LIN {X 0,Y 299.313,Z 470.406,A -85,B 0,C 180,E1 -16726.074,E2 -16726.074} C_VEL
LIN {X 0,Y 297.417,Z 475.338,A -85,B 0,C 180,E1 -16727.721,E2 -16727.721} C_VEL
LIN {X 0,Y 295.4,Z 479.817,A -85,B 0,C 180,E1 -16729.721,E2 -16729.721} C_VEL
LIN {X 0,Y 293.632,Z 482.84,A -85,B 0,C 180,E1 -16731.743,E2 -16731.743} C_VEL
LIN {X 0,Y 292.623,Z 484.058,A -85,B 0,C 180,E1 -16733.103,E2 -16733.103} C_VEL
LIN {X 0,Y 291.792,Z 484.661,A -85,B 0,C 180,E1 -16734.471,E2 -16734.471} C_VEL
LIN {X 0,Y 291.126,Z 484.675,A -85,B 0,C 180,E1 -16735.847,E2 -16735.847} C_VEL
LIN {X 0,Y 290.687,Z 484.067,A -85,B 0,C 180,E1 -16737.229,E2 -16737.229} C_VEL
LIN {X 0,Y 290.38,Z 482.836,A -85,B 0,C 180,E1 -16738.613,E2 -16738.613} C_VEL
LIN {X 0,Y 290.157,Z 479.788,A -85,B 0,C 180,E1 -16740.694,E2 -16740.694} C_VEL
LIN {X 0,Y 290.14,Z 475.202,A -85,B 0,C 180,E1 -16742.777,E2 -16742.777} C_VEL
LIN {X 0,Y 290.478,Z 468.838,A -85,B 0,C 180,E1 -16744.858,E2 -16744.858} C_VEL
LIN {X 0,Y 290.817,Z 461.925,A -85,B 0,C 180,E1 -16746.592,E2 -16746.592} C_VEL
LIN {X 0,Y 291.139,Z 453.117,A -85,B 0,C 180,E1 -16748.328,E2 -16748.328} C_VEL
LIN {X 0,Y 291.598,Z 443.01,A -85,B 0,C 180,E1 -16749.888,E2 -16749.888} C_VEL
LIN {X 0,Y 292.119,Z 433.031,A -85,B 0,C 180,E1 -16751.097,E2 -16751.097} C_VEL
LIN {X 0,Y 290.871,Z 421.3,A -85,B 0,C 180,E1 -16752.206,E2 -16752.206} C_VEL
LIN {X 0,Y 290.218,Z 413.705,A -85,B 0,C 180,E1 -16752.766,E2 -16752.766} C_VEL
LIN {X 0,Y 290.434,Z 407.138,A -85,B 0,C 180,E1 -16756.881,E2 -16756.881} C_VEL
LIN {X 0,Y 290.756,Z 401.449,A -85,B 0,C 180,E1 -16760.517,E2 -16760.517} C_VEL
LIN {X 0,Y 291.158,Z 394.62,A -85,B 0,C 180,E1 -16764.987,E2 -16764.987} C_VEL
LIN {X 0,Y 291.612,Z 388.864,A -85,B 0,C 180,E1 -16768.817,E2 -16768.817} C_VEL
LIN {X 0,Y 291.797,Z 385.393,A -85,B 0,C 180,E1 -16771.187,E2 -16771.187} C_VEL
LIN {X 0,Y 291.576,Z 384.166,A -85,B 0,C 180,E1 -16772.181,E2 -16772.181} C_VEL
LIN {X 0,Y 291.408,Z 384.187,A -85,B 0,C 180,E1 -16777.081,E2 -16777.081} C_VEL
LIN {X 0,Y 291.335,Z 384.196,A -85,B 0,C 180,E1 -16780.642,E2 -16780.642} C_VEL
LIN {X 0,Y 291.316,Z 384.196,A -85,B 0,C 180,E1 -16784.397,E2 -16784.397} C_VEL
LIN {X 0,Y 291.33,Z 384.196,A -85,B 0,C 180,E1 -16788.404,E2 -16788.404} C_VEL
LIN {X 0,Y 291.35,Z 384.191,A -85,B 0,C 180,E1 -16791.158,E2 -16791.158} C_VEL
LIN {X 0,Y 291.364,Z 384.194,A -85,B 0,C 180,E1 -16794.626,E2 -16794.626} C_VEL
LIN {X 0,Y 291.373,Z 384.188,A -85,B 0,C 180,E1 -16797.951,E2 -16797.951} C_VEL
LIN {X 0,Y 291.38,Z 384.187,A -85,B 0,C 180,E1 -16801.158,E2 -16801.158} C_VEL
LIN {X 0,Y 291.418,Z 384.186,A -85,B 0,C 180,E1 -16804.272,E2 -16804.272} C_VEL
LIN {X 0,Y 291.392,Z 384.185,A -85,B 0,C 180,E1 -16807.3,E2 -16807.3} C_VEL
LIN {X 0,Y 291.462,Z 384.18,A -85,B 0,C 180,E1 -16810.27,E2 -16810.27} C_VEL
LIN {X 0,Y 291.558,Z 384.166,A -85,B 0,C 180,E1 -16814.624,E2 -16814.624} C_VEL
LIN {X 0,Y 291.539,Z 384.167,A -85,B 0,C 180,E1 -16818.881,E2 -16818.881} C_VEL
LIN {X 0,Y 291.691,Z 384.15,A -85,B 0,C 180,E1 -16821.688,E2 -16821.688} C_VEL
LIN {X 0,Y 291.63,Z 384.157,A -85,B 0,C 180,E1 -16824.468,E2 -16824.468} C_VEL
LIN {X 0,Y 291.892,Z 384.124,A -85,B 0,C 180,E1 -16828.62,E2 -16828.62} C_VEL
LIN {X 0,Y 291.894,Z 384.124,A -85,B 0,C 180,E1 -16831.38,E2 -16831.38} C_VEL
LIN {X 0,Y 291.745,Z 384.141,A -85,B 0,C 180,E1 -16836.918,E2 -16836.918} C_VEL
LIN {X 0,Y 291.632,Z 384.159,A -85,B 0,C 180,E1 -16839.712,E2 -16839.712} C_VEL
LIN {X 0,Y 291.525,Z 384.172,A -85,B 0,C 180,E1 -16843.95,E2 -16843.95} C_VEL
LIN {X 0,Y 291.49,Z 384.173,A -85,B 0,C 180,E1 -16846.818,E2 -16846.818} C_VEL
LIN {X 0,Y 291.454,Z 384.18,A -85,B 0,C 180,E1 -16849.875,E2 -16849.875} C_VEL
LIN {X 0,Y 291.403,Z 384.185,A -85,B 0,C 180,E1 -16854.205,E2 -16854.205} C_VEL
LIN {X 0,Y 291.422,Z 384.184,A -85,B 0,C 180,E1 -16857.272,E2 -16857.272} C_VEL
LIN {X 0,Y 291.336,Z 384.191,A -85,B 0,C 180,E1 -16860.437,E2 -16860.437} C_VEL
LIN {X 0,Y 291.347,Z 384.194,A -85,B 0,C 180,E1 -16863.698,E2 -16863.698} C_VEL
LIN {X 0,Y 291.397,Z 384.188,A -85,B 0,C 180,E1 -16867.259,E2 -16867.259} C_VEL
LIN {X 0,Y 291.336,Z 384.192,A -85,B 0,C 180,E1 -16870.642,E2 -16870.642} C_VEL
LIN {X 0,Y 291.291,Z 384.198,A -85,B 0,C 180,E1 -16874.402,E2 -16874.402} C_VEL
LIN {X 0,Y 291.328,Z 384.193,A -85,B 0,C 180,E1 -16878.404,E2 -16878.404} C_VEL
LIN {X 0,Y 291.35,Z 384.196,A -85,B 0,C 180,E1 -16881.157,E2 -16881.157} C_VEL
LIN {X 0,Y 291.362,Z 384.19,A -85,B 0,C 180,E1 -16884.626,E2 -16884.626} C_VEL
LIN {X 0,Y 291.374,Z 384.187,A -85,B 0,C 180,E1 -16887.951,E2 -16887.951} C_VEL
LIN {X 0,Y 291.385,Z 384.189,A -85,B 0,C 180,E1 -16891.158,E2 -16891.158} C_VEL
LIN {X 0,Y 291.418,Z 384.182,A -85,B 0,C 180,E1 -16894.272,E2 -16894.272} C_VEL
LIN {X 0,Y 291.384,Z 384.188,A -85,B 0,C 180,E1 -16897.3,E2 -16897.3} C_VEL
LIN {X 0,Y 291.46,Z 384.178,A -85,B 0,C 180,E1 -16900.27,E2 -16900.27} C_VEL
LIN {X 0,Y 291.557,Z 384.168,A -85,B 0,C 180,E1 -16904.624,E2 -16904.624} C_VEL
LIN {X 0,Y 291.541,Z 384.17,A -85,B 0,C 180,E1 -16908.881,E2 -16908.881} C_VEL
LIN {X 0,Y 291.711,Z 384.144,A -85,B 0,C 180,E1 -16911.688,E2 -16911.688} C_VEL
LIN {X 0,Y 291.633,Z 384.159,A -85,B 0,C 180,E1 -16914.468,E2 -16914.468} C_VEL
LIN {X 0,Y 291.892,Z 384.126,A -85,B 0,C 180,E1 -16918.62,E2 -16918.62} C_VEL
LIN {X 0,Y 291.895,Z 384.122,A -85,B 0,C 180,E1 -16921.38,E2 -16921.38} C_VEL
LIN {X 0,Y 291.749,Z 384.141,A -85,B 0,C 180,E1 -16926.918,E2 -16926.918} C_VEL
LIN {X 0,Y 291.631,Z 384.155,A -85,B 0,C 180,E1 -16929.712,E2 -16929.712} C_VEL
LIN {X 0,Y 291.502,Z 384.172,A -85,B 0,C 180,E1 -16933.035,E2 -16933.035} C_VEL
LIN {X 0,Y 290.827,Z 384.26,A -85,B 0,C 180,E1 -16934.188,E2 -16934.188} C_VEL
LIN {X 0,Y 287.966,Z 384.615,A -85,B 0,C 180,E1 -16936.065,E2 -16936.065} C_VEL
LIN {X 0,Y 285.533,Z 384.917,A -85,B 0,C 180,E1 -16937.589,E2 -16937.589} C_VEL
LIN {X 0,Y 284.476,Z 385.048,A -85,B 0,C 180,E1 -16938.77,E2 -16938.77} C_VEL
LIN {X 0,Y 284.383,Z 385.058,A -85,B 0,C 180,E1 -16939.171,E2 -16939.171} C_VEL
LIN {X 0,Y 284.371,Z 385.063,A -85,B 0,C 180,E1 -16943.875,E2 -16943.875} C_VEL
LIN {X 0,Y 284.397,Z 385.056,A -85,B 0,C 180,E1 -16947.173,E2 -16947.173} C_VEL
LIN {X 0,Y 284.295,Z 385.07,A -85,B 0,C 180,E1 -16951.274,E2 -16951.274} C_VEL
LIN {X 0,Y 284.363,Z 385.061,A -85,B 0,C 180,E1 -16955.354,E2 -16955.354} C_VEL
LIN {X 0,Y 284.325,Z 385.068,A -85,B 0,C 180,E1 -16958.167,E2 -16958.167} C_VEL
LIN {X 0,Y 284.271,Z 385.073,A -85,B 0,C 180,E1 -16962.125,E2 -16962.125} C_VEL
LIN {X 0,Y 284.287,Z 385.073,A -85,B 0,C 180,E1 -16966.195,E2 -16966.195} C_VEL
LIN {X 0,Y 284.354,Z 385.245,A -85,B 0,C 180,E1 -16968.499,E2 -16968.499} C_VEL
LIN {X 0,Y 286.142,Z 394.145,A -85,B 0,C 180,E1 -16972.563,E2 -16972.563} C_VEL
LIN {X 0,Y 288.209,Z 404.002,A -85,B 0,C 180,E1 -16976.866,E2 -16976.866} C_VEL
LIN {X 0,Y 289.225,Z 409.855,A -85,B 0,C 180,E1 -16979.317,E2 -16979.317} C_VEL
LIN {X 0,Y 286.887,Z 421.364,A -85,B 0,C 180,E1 -16983.835,E2 -16983.835} C_VEL
LIN {X 0,Y 284.814,Z 434.601,A -85,B 0,C 180,E1 -16989.035,E2 -16989.035} C_VEL
LIN {X 0,Y 284.356,Z 438.709,A -85,B 0,C 180,E1 -16990.65,E2 -16990.65} C_VEL
LIN {X 0,Y 284.635,Z 450.827,A -85,B 0,C 180,E1 -16991.277,E2 -16991.277} C_VEL
LIN {X 0,Y 285.426,Z 463.008,A -85,B 0,C 180,E1 -16992.167,E2 -16992.167} C_VEL
LIN {X 0,Y 286.069,Z 473.069,A -85,B 0,C 180,E1 -16993.126,E2 -16993.126} C_VEL
LIN {X 0,Y 285.367,Z 484.226,A -85,B 0,C 180,E1 -16994.465,E2 -16994.465} C_VEL
LIN {X 0,Y 284.62,Z 493.685,A -85,B 0,C 180,E1 -16995.887,E2 -16995.887} C_VEL
LIN {X 0,Y 284.078,Z 502.385,A -85,B 0,C 180,E1 -16997.498,E2 -16997.498} C_VEL
LIN {X 0,Y 283.619,Z 510.299,A -85,B 0,C 180,E1 -16999.289,E2 -16999.289} C_VEL
LIN {X 0,Y 283.365,Z 517.923,A -85,B 0,C 180,E1 -17001.442,E2 -17001.442} C_VEL
LIN {X 0,Y 283.392,Z 524.403,A -85,B 0,C 180,E1 -17003.804,E2 -17003.804} C_VEL
LIN {X 0,Y 283.412,Z 528.421,A -85,B 0,C 180,E1 -17005.734,E2 -17005.734} C_VEL
LIN {X 0,Y 283.463,Z 530.725,A -85,B 0,C 180,E1 -17007.158,E2 -17007.158} C_VEL
LIN {X 0,Y 283.429,Z 532.5,A -85,B 0,C 180,E1 -17008.579,E2 -17008.579} C_VEL
LIN {X 0,Y 283.353,Z 533.796,A -85,B 0,C 180,E1 -17010,E2 -17010} C_VEL
LIN {X 0,Y 283.316,Z 534.601,A -85,B 0,C 180,E1 -17011.422,E2 -17011.422} C_VEL
LIN {X 0,Y 283.067,Z 534.958,A -85,B 0,C 180,E1 -17012.846,E2 -17012.846} C_VEL
LIN {X 0,Y 282.807,Z 534.888,A -85,B 0,C 180,E1 -17014.276,E2 -17014.276} C_VEL
LIN {X 0,Y 282.714,Z 534.18,A -85,B 0,C 180,E1 -17016.087,E2 -17016.087} C_VEL
LIN {X 0,Y 282.793,Z 532.167,A -85,B 0,C 180,E1 -17018.576,E2 -17018.576} C_VEL
LIN {X 0,Y 283.348,Z 528.257,A -85,B 0,C 180,E1 -17021.445,E2 -17021.445} C_VEL
LIN {X 0,Y 284.44,Z 524.2,A -85,B 0,C 180,E1 -17023.576,E2 -17023.576} C_VEL
LIN {X 0,Y 285.821,Z 519.069,A -85,B 0,C 180,E1 -17025.693,E2 -17025.693} C_VEL
LIN {X 0,Y 288.032,Z 511.787,A -85,B 0,C 180,E1 -17028.043,E2 -17028.043} C_VEL
LIN {X 0,Y 290.656,Z 503.511,A -85,B 0,C 180,E1 -17030.155,E2 -17030.155} C_VEL
LIN {X 0,Y 293.667,Z 493.625,A -85,B 0,C 180,E1 -17032.144,E2 -17032.144} C_VEL
LIN {X 0,Y 296.144,Z 484.696,A -85,B 0,C 180,E1 -17033.608,E2 -17033.608} C_VEL
LIN {X 0,Y 297.823,Z 474.304,A -85,B 0,C 180,E1 -17035.136,E2 -17035.136} C_VEL
LIN {X 0,Y 298.035,Z 463.954,A -85,B 0,C 180,E1 -17036.618,E2 -17036.618} C_VEL
LIN {X 0,Y 297.261,Z 453.783,A -85,B 0,C 180,E1 -17038.065,E2 -17038.065} C_VEL
LIN {X 0,Y 295.282,Z 442.412,A -85,B 0,C 180,E1 -17039.714,E2 -17039.714} C_VEL
LIN {X 0,Y 293.524,Z 434.527,A -85,B 0,C 180,E1 -17040.894,E2 -17040.894} C_VEL
LIN {X 0,Y 294.835,Z 431.545,A -85,B 0,C 180,E1 -17042.435,E2 -17042.435} C_VEL
LIN {X 0,Y 295.09,Z 429.766,A -85,B 0,C 180,E1 -17043.532,E2 -17043.532} C_VEL
LIN {X 0,Y 294.427,Z 425.778,A -85,B 0,C 180,E1 -17046.638,E2 -17046.638} C_VEL
LIN {X 0,Y 293.633,Z 422.199,A -85,B 0,C 180,E1 -17050.259,E2 -17050.259} C_VEL
LIN {X 0,Y 293.026,Z 419.56,A -85,B 0,C 180,E1 -17054.071,E2 -17054.071} C_VEL
LIN {X 0,Y 292.456,Z 418.155,A -85,B 0,C 180,E1 -17057.711,E2 -17057.711} C_VEL
LIN {X 0,Y 292.088,Z 417.72,A -85,B 0,C 180,E1 -17061.274,E2 -17061.274} C_VEL
LIN {X 0,Y 291.76,Z 418.132,A -85,B 0,C 180,E1 -17064.682,E2 -17064.682} C_VEL
LIN {X 0,Y 291.278,Z 419.282,A -85,B 0,C 180,E1 -17067.939,E2 -17067.939} C_VEL
LIN {X 0,Y 290.309,Z 421.098,A -85,B 0,C 180,E1 -17071.042,E2 -17071.042} C_VEL
LIN {X 0,Y 289.414,Z 422.981,A -85,B 0,C 180,E1 -17073.484,E2 -17073.484} C_VEL
LIN {X 0,Y 290.356,Z 425.753,A -85,B 0,C 180,E1 -17074.171,E2 -17074.171} C_VEL
LIN {X 0,Y 292.047,Z 429.532,A -85,B 0,C 180,E1 -17075.232,E2 -17075.232} C_VEL
LIN {X 0,Y 294.97,Z 437.823,A -85,B 0,C 180,E1 -17077.353,E2 -17077.353} C_VEL
LIN {X 0,Y 297.063,Z 446.831,A -85,B 0,C 180,E1 -17079.51,E2 -17079.51} C_VEL
LIN {X 0,Y 297.877,Z 454.634,A -85,B 0,C 180,E1 -17081.366,E2 -17081.366} C_VEL
LIN {X 0,Y 297.878,Z 457.869,A -85,B 0,C 180,E1 -17082.139,E2 -17082.139} C_VEL
LIN {X 0,Y 295.496,Z 465.423,A -85,B 0,C 180,E1 -17083.772,E2 -17083.772} C_VEL
LIN {X 0,Y 292.703,Z 472.611,A -85,B 0,C 180,E1 -17085.753,E2 -17085.753} C_VEL
LIN {X 0,Y 290.705,Z 477.27,A -85,B 0,C 180,E1 -17087.433,E2 -17087.433} C_VEL
LIN {X 0,Y 288.587,Z 481.379,A -85,B 0,C 180,E1 -17089.476,E2 -17089.476} C_VEL
LIN {X 0,Y 286.711,Z 484.087,A -85,B 0,C 180,E1 -17091.543,E2 -17091.543} C_VEL
LIN {X 0,Y 285.658,Z 485.145,A -85,B 0,C 180,E1 -17092.934,E2 -17092.934} C_VEL
LIN {X 0,Y 284.788,Z 485.597,A -85,B 0,C 180,E1 -17094.335,E2 -17094.335} C_VEL
LIN {X 0,Y 284.107,Z 485.431,A -85,B 0,C 180,E1 -17095.744,E2 -17095.744} C_VEL
LIN {X 0,Y 283.625,Z 484.644,A -85,B 0,C 180,E1 -17097.159,E2 -17097.159} C_VEL
LIN {X 0,Y 283.202,Z 482.309,A -85,B 0,C 180,E1 -17099.289,E2 -17099.289} C_VEL
LIN {X 0,Y 283.014,Z 478.516,A -85,B 0,C 180,E1 -17101.423,E2 -17101.423} C_VEL
LIN {X 0,Y 283.138,Z 473.111,A -85,B 0,C 180,E1 -17103.558,E2 -17103.558} C_VEL
LIN {X 0,Y 283.491,Z 467.218,A -85,B 0,C 180,E1 -17105.334,E2 -17105.334} C_VEL
LIN {X 0,Y 283.77,Z 459.657,A -85,B 0,C 180,E1 -17107.113,E2 -17107.113} C_VEL
LIN {X 0,Y 284.156,Z 451.106,A -85,B 0,C 180,E1 -17108.713,E2 -17108.713} C_VEL
LIN {X 0,Y 284.552,Z 441.577,A -85,B 0,C 180,E1 -17110.136,E2 -17110.136} C_VEL
LIN {X 0,Y 284.985,Z 432.735,A -85,B 0,C 180,E1 -17111.198,E2 -17111.198} C_VEL
LIN {X 0,Y 283.812,Z 421.87,A -85,B 0,C 180,E1 -17112.242,E2 -17112.242} C_VEL
LIN {X 0,Y 283.147,Z 414,A -85,B 0,C 180,E1 -17112.863,E2 -17112.863} C_VEL
LIN {X 0,Y 283.379,Z 407.027,A -85,B 0,C 180,E1 -17117.314,E2 -17117.314} C_VEL
LIN {X 0,Y 283.713,Z 401.294,A -85,B 0,C 180,E1 -17121.051,E2 -17121.051} C_VEL
LIN {X 0,Y 284.077,Z 395.554,A -85,B 0,C 180,E1 -17124.871,E2 -17124.871} C_VEL
LIN {X 0,Y 284.548,Z 389.768,A -85,B 0,C 180,E1 -17128.792,E2 -17128.792} C_VEL
LIN {X 0,Y 284.772,Z 386.274,A -85,B 0,C 180,E1 -17131.216,E2 -17131.216} C_VEL
LIN {X 0,Y 284.524,Z 385.044,A -85,B 0,C 180,E1 -17132.269,E2 -17132.269} C_VEL
LIN {X 0,Y 284.343,Z 385.064,A -85,B 0,C 180,E1 -17136.385,E2 -17136.385} C_VEL
LIN {X 0,Y 284.308,Z 385.068,A -85,B 0,C 180,E1 -17139.995,E2 -17139.995} C_VEL
LIN {X 0,Y 284.268,Z 385.073,A -85,B 0,C 180,E1 -17144.195,E2 -17144.195} C_VEL
LIN {X 0,Y 284.275,Z 385.073,A -85,B 0,C 180,E1 -17148.125,E2 -17148.125} C_VEL
LIN {X 0,Y 284.322,Z 385.067,A -85,B 0,C 180,E1 -17152.279,E2 -17152.279} C_VEL
LIN {X 0,Y 284.311,Z 385.068,A -85,B 0,C 180,E1 -17155.351,E2 -17155.351} C_VEL
LIN {X 0,Y 284.296,Z 385.071,A -85,B 0,C 180,E1 -17158.726,E2 -17158.726} C_VEL
LIN {X 0,Y 284.398,Z 385.058,A -85,B 0,C 180,E1 -17162.827,E2 -17162.827} C_VEL
LIN {X 0,Y 284.372,Z 385.061,A -85,B 0,C 180,E1 -17166.707,E2 -17166.707} C_VEL
LIN {X 0,Y 284.407,Z 385.055,A -85,B 0,C 180,E1 -17171.262,E2 -17171.262} C_VEL
LIN {X 0,Y 284.495,Z 385.047,A -85,B 0,C 180,E1 -17174.459,E2 -17174.459} C_VEL
LIN {X 0,Y 284.491,Z 385.046,A -85,B 0,C 180,E1 -17178.601,E2 -17178.601} C_VEL
LIN {X 0,Y 284.642,Z 385.027,A -85,B 0,C 180,E1 -17181.48,E2 -17181.48} C_VEL
LIN {X 0,Y 284.6,Z 385.033,A -85,B 0,C 180,E1 -17184.331,E2 -17184.331} C_VEL
LIN {X 0,Y 284.858,Z 385,A -85,B 0,C 180,E1 -17188.586,E2 -17188.586} C_VEL
LIN {X 0,Y 284.859,Z 385,A -85,B 0,C 180,E1 -17191.414,E2 -17191.414} C_VEL
LIN {X 0,Y 284.697,Z 385.019,A -85,B 0,C 180,E1 -17197.09,E2 -17197.09} C_VEL
LIN {X 0,Y 284.57,Z 385.039,A -85,B 0,C 180,E1 -17199.955,E2 -17199.955} C_VEL
LIN {X 0,Y 284.485,Z 385.046,A -85,B 0,C 180,E1 -17204.303,E2 -17204.303} C_VEL
LIN {X 0,Y 284.429,Z 385.054,A -85,B 0,C 180,E1 -17207.248,E2 -17207.248} C_VEL
LIN {X 0,Y 284.384,Z 385.058,A -85,B 0,C 180,E1 -17210.242,E2 -17210.242} C_VEL
LIN {X 0,Y 284.372,Z 385.062,A -85,B 0,C 180,E1 -17213.875,E2 -17213.875} C_VEL
LIN {X 0,Y 284.397,Z 385.059,A -85,B 0,C 180,E1 -17217.173,E2 -17217.173} C_VEL
LIN {X 0,Y 284.296,Z 385.071,A -85,B 0,C 180,E1 -17221.274,E2 -17221.274} C_VEL
LIN {X 0,Y 284.364,Z 385.065,A -85,B 0,C 180,E1 -17225.354,E2 -17225.354} C_VEL
LIN {X 0,Y 284.325,Z 385.064,A -85,B 0,C 180,E1 -17228.167,E2 -17228.167} C_VEL
LIN {X 0,Y 284.271,Z 385.072,A -85,B 0,C 180,E1 -17232.124,E2 -17232.124} C_VEL
LIN {X 0,Y 284.256,Z 385.073,A -85,B 0,C 180,E1 -17236.189,E2 -17236.189} C_VEL
LIN {X 0,Y 284.308,Z 385.068,A -85,B 0,C 180,E1 -17240.024,E2 -17240.024} C_VEL
LIN {X 0,Y 284.332,Z 385.065,A -85,B 0,C 180,E1 -17243.614,E2 -17243.614} C_VEL
LIN {X 0,Y 284.309,Z 385.071,A -85,B 0,C 180,E1 -17247.189,E2 -17247.189} C_VEL
LIN {X 0,Y 284.361,Z 385.062,A -85,B 0,C 180,E1 -17250.376,E2 -17250.376} C_VEL
LIN {X 0,Y 284.38,Z 385.058,A -85,B 0,C 180,E1 -17253.587,E2 -17253.587} C_VEL
LIN {X 0,Y 284.368,Z 385.063,A -85,B 0,C 180,E1 -17256.707,E2 -17256.707} C_VEL
LIN {X 0,Y 284.406,Z 385.056,A -85,B 0,C 180,E1 -17261.262,E2 -17261.262} C_VEL
LIN {X 0,Y 284.494,Z 385.046,A -85,B 0,C 180,E1 -17264.459,E2 -17264.459} C_VEL
LIN {X 0,Y 284.492,Z 385.049,A -85,B 0,C 180,E1 -17268.601,E2 -17268.601} C_VEL
LIN {X 0,Y 284.661,Z 385.023,A -85,B 0,C 180,E1 -17271.481,E2 -17271.481} C_VEL
LIN {X 0,Y 284.603,Z 385.033,A -85,B 0,C 180,E1 -17274.331,E2 -17274.331} C_VEL
LIN {X 0,Y 284.858,Z 385.003,A -85,B 0,C 180,E1 -17278.586,E2 -17278.586} C_VEL
LIN {X 0,Y 284.861,Z 384.998,A -85,B 0,C 180,E1 -17281.414,E2 -17281.414} C_VEL
LIN {X 0,Y 284.701,Z 385.018,A -85,B 0,C 180,E1 -17287.09,E2 -17287.09} C_VEL
LIN {X 0,Y 284.568,Z 385.036,A -85,B 0,C 180,E1 -17289.955,E2 -17289.955} C_VEL
LIN {X 0,Y 284.483,Z 385.05,A -85,B 0,C 180,E1 -17294.303,E2 -17294.303} C_VEL
LIN {X 0,Y 284.427,Z 385.051,A -85,B 0,C 180,E1 -17297.248,E2 -17297.248} C_VEL
LIN {X 0,Y 284.383,Z 385.058,A -85,B 0,C 180,E1 -17299.171,E2 -17299.171} C_VEL
LIN {X 0,Y 283.684,Z 385.149,A -85,B 0,C 180,E1 -17300.352,E2 -17300.352} C_VEL
LIN {X 0,Y 280.793,Z 385.509,A -85,B 0,C 180,E1 -17302.275,E2 -17302.275} C_VEL
LIN {X 0,Y 278.377,Z 385.809,A -85,B 0,C 180,E1 -17303.837,E2 -17303.837} C_VEL
LIN {X 0,Y 277.376,Z 385.93,A -85,B 0,C 180,E1 -17305.048,E2 -17305.048} C_VEL
LIN {X 0,Y 277.312,Z 385.939,A -85,B 0,C 180,E1 -17305.458,E2 -17305.458} C_VEL
LIN {X 0,Y 277.27,Z 385.945,A -85,B 0,C 180,E1 -17308.79,E2 -17308.79} C_VEL
LIN {X 0,Y 277.245,Z 385.95,A -85,B 0,C 180,E1 -17312.164,E2 -17312.164} C_VEL
LIN {X 0,Y 277.326,Z 385.94,A -85,B 0,C 180,E1 -17315.811,E2 -17315.811} C_VEL
LIN {X 0,Y 277.239,Z 385.95,A -85,B 0,C 180,E1 -17319.327,E2 -17319.327} C_VEL
LIN {X 0,Y 277.218,Z 385.95,A -85,B 0,C 180,E1 -17323.196,E2 -17323.196} C_VEL
LIN {X 0,Y 277.242,Z 385.951,A -85,B 0,C 180,E1 -17327.319,E2 -17327.319} C_VEL
LIN {X 0,Y 277.278,Z 386.029,A -85,B 0,C 180,E1 -17328.123,E2 -17328.123} C_VEL
LIN {X 0,Y 279.014,Z 394.549,A -85,B 0,C 180,E1 -17332.151,E2 -17332.151} C_VEL
LIN {X 0,Y 281.067,Z 404.492,A -85,B 0,C 180,E1 -17336.626,E2 -17336.626} C_VEL
LIN {X 0,Y 282.099,Z 409.701,A -85,B 0,C 180,E1 -17338.872,E2 -17338.872} C_VEL
LIN {X 0,Y 281.705,Z 412.618,A -85,B 0,C 180,E1 -17340.069,E2 -17340.069} C_VEL
LIN {X 0,Y 279.253,Z 424.679,A -85,B 0,C 180,E1 -17344.961,E2 -17344.961} C_VEL
LIN {X 0,Y 277.296,Z 438.45,A -85,B 0,C 180,E1 -17350.552,E2 -17350.552} C_VEL
LIN {X 0,Y 277.6,Z 451.579,A -85,B 0,C 180,E1 -17351.264,E2 -17351.264} C_VEL
LIN {X 0,Y 278.381,Z 464.396,A -85,B 0,C 180,E1 -17352.27,E2 -17352.27} C_VEL
LIN {X 0,Y 278.958,Z 473.683,A -85,B 0,C 180,E1 -17353.209,E2 -17353.209} C_VEL
LIN {X 0,Y 278.218,Z 484.829,A -85,B 0,C 180,E1 -17354.619,E2 -17354.619} C_VEL
LIN {X 0,Y 277.415,Z 496.092,A -85,B 0,C 180,E1 -17356.447,E2 -17356.447} C_VEL
LIN {X 0,Y 276.82,Z 505.041,A -85,B 0,C 180,E1 -17358.281,E2 -17358.281} C_VEL
LIN {X 0,Y 276.406,Z 513.642,A -85,B 0,C 180,E1 -17360.487,E2 -17360.487} C_VEL
LIN {X 0,Y 276.336,Z 520.358,A -85,B 0,C 180,E1 -17362.694,E2 -17362.694} C_VEL
LIN {X 0,Y 276.407,Z 525.569,A -85,B 0,C 180,E1 -17364.894,E2 -17364.894} C_VEL
LIN {X 0,Y 276.438,Z 529.435,A -85,B 0,C 180,E1 -17367.086,E2 -17367.086} C_VEL
LIN {X 0,Y 276.414,Z 531.309,A -85,B 0,C 180,E1 -17368.543,E2 -17368.543} C_VEL
LIN {X 0,Y 276.337,Z 532.697,A -85,B 0,C 180,E1 -17370,E2 -17370} C_VEL
LIN {X 0,Y 276.27,Z 533.632,A -85,B 0,C 180,E1 -17371.458,E2 -17371.458} C_VEL
LIN {X 0,Y 276.002,Z 534.059,A -85,B 0,C 180,E1 -17372.919,E2 -17372.919} C_VEL
LIN {X 0,Y 275.662,Z 533.702,A -85,B 0,C 180,E1 -17375.853,E2 -17375.853} C_VEL
LIN {X 0,Y 275.739,Z 531.663,A -85,B 0,C 180,E1 -17378.797,E2 -17378.797} C_VEL
LIN {X 0,Y 276.136,Z 529.08,A -85,B 0,C 180,E1 -17381.005,E2 -17381.005} C_VEL
LIN {X 0,Y 277.089,Z 525.55,A -85,B 0,C 180,E1 -17383.196,E2 -17383.196} C_VEL
LIN {X 0,Y 278.489,Z 521.009,A -85,B 0,C 180,E1 -17385.366,E2 -17385.366} C_VEL
LIN {X 0,Y 280.29,Z 515.367,A -85,B 0,C 180,E1 -17387.511,E2 -17387.511} C_VEL
LIN {X 0,Y 282.669,Z 508.402,A -85,B 0,C 180,E1 -17389.612,E2 -17389.612} C_VEL
LIN {X 0,Y 285.542,Z 499.934,A -85,B 0,C 180,E1 -17391.666,E2 -17391.666} C_VEL
LIN {X 0,Y 288.405,Z 491.409,A -85,B 0,C 180,E1 -17393.328,E2 -17393.328} C_VEL
LIN {X 0,Y 290.779,Z 482.358,A -85,B 0,C 180,E1 -17394.831,E2 -17394.831} C_VEL
LIN {X 0,Y 292.085,Z 473.699,A -85,B 0,C 180,E1 -17396.17,E2 -17396.17} C_VEL
LIN {X 0,Y 292.37,Z 464.469,A -85,B 0,C 180,E1 -17397.592,E2 -17397.592} C_VEL
LIN {X 0,Y 291.554,Z 453.535,A -85,B 0,C 180,E1 -17399.272,E2 -17399.272} C_VEL
LIN {X 0,Y 290.079,Z 443.83,A -85,B 0,C 180,E1 -17400.805,E2 -17400.805} C_VEL
LIN {X 0,Y 287.962,Z 433.94,A -85,B 0,C 180,E1 -17402.475,E2 -17402.475} C_VEL
LIN {X 0,Y 288.346,Z 432.677,A -85,B 0,C 180,E1 -17403.219,E2 -17403.219} C_VEL
LIN {X 0,Y 287.967,Z 429.199,A -85,B 0,C 180,E1 -17405.855,E2 -17405.855} C_VEL
LIN {X 0,Y 287.14,Z 425.414,A -85,B 0,C 180,E1 -17409.522,E2 -17409.522} C_VEL
LIN {X 0,Y 286.591,Z 423.048,A -85,B 0,C 180,E1 -17412.635,E2 -17412.635} C_VEL
LIN {X 0,Y 286.182,Z 421.547,A -85,B 0,C 180,E1 -17415.413,E2 -17415.413} C_VEL
LIN {X 0,Y 285.748,Z 420.614,A -85,B 0,C 180,E1 -17418.389,E2 -17418.389} C_VEL
LIN {X 0,Y 285.589,Z 420.315,A -85,B 0,C 180,E1 -17420.221,E2 -17420.221} C_VEL
LIN {X 0,Y 285.211,Z 420.458,A -85,B 0,C 180,E1 -17423.744,E2 -17423.744} C_VEL
LIN {X 0,Y 284.722,Z 421.363,A -85,B 0,C 180,E1 -17427.109,E2 -17427.109} C_VEL
LIN {X 0,Y 283.806,Z 423.003,A -85,B 0,C 180,E1 -17430.313,E2 -17430.313} C_VEL
LIN {X 0,Y 283.371,Z 423.811,A -85,B 0,C 180,E1 -17431.533,E2 -17431.533} C_VEL
LIN {X 0,Y 284.386,Z 426.78,A -85,B 0,C 180,E1 -17432.395,E2 -17432.395} C_VEL
LIN {X 0,Y 285.663,Z 429.586,A -85,B 0,C 180,E1 -17433.32,E2 -17433.32} C_VEL
LIN {X 0,Y 288.026,Z 435.893,A -85,B 0,C 180,E1 -17435.184,E2 -17435.184} C_VEL
LIN {X 0,Y 290.158,Z 443.293,A -85,B 0,C 180,E1 -17437.198,E2 -17437.198} C_VEL
LIN {X 0,Y 291.474,Z 450.903,A -85,B 0,C 180,E1 -17439.167,E2 -17439.167} C_VEL
LIN {X 0,Y 291.947,Z 457.95,A -85,B 0,C 180,E1 -17440.973,E2 -17440.973} C_VEL
LIN {X 0,Y 291.658,Z 460.997,A -85,B 0,C 180,E1 -17441.744,E2 -17441.744} C_VEL
LIN {X 0,Y 289.034,Z 468.123,A -85,B 0,C 180,E1 -17443.399,E2 -17443.399} C_VEL
LIN {X 0,Y 286.572,Z 473.846,A -85,B 0,C 180,E1 -17445.078,E2 -17445.078} C_VEL
LIN {X 0,Y 283.973,Z 479.115,A -85,B 0,C 180,E1 -17447.13,E2 -17447.13} C_VEL
LIN {X 0,Y 281.77,Z 482.93,A -85,B 0,C 180,E1 -17449.218,E2 -17449.218} C_VEL
LIN {X 0,Y 279.81,Z 485.35,A -85,B 0,C 180,E1 -17451.332,E2 -17451.332} C_VEL
LIN {X 0,Y 278.69,Z 486.197,A -85,B 0,C 180,E1 -17452.756,E2 -17452.756} C_VEL
LIN {X 0,Y 277.781,Z 486.458,A -85,B 0,C 180,E1 -17454.192,E2 -17454.192} C_VEL
LIN {X 0,Y 277.089,Z 486.122,A -85,B 0,C 180,E1 -17455.636,E2 -17455.636} C_VEL
LIN {X 0,Y 276.566,Z 485.18,A -85,B 0,C 180,E1 -17457.087,E2 -17457.087} C_VEL
LIN {X 0,Y 276.131,Z 482.601,A -85,B 0,C 180,E1 -17459.271,E2 -17459.271} C_VEL
LIN {X 0,Y 275.916,Z 478.548,A -85,B 0,C 180,E1 -17461.46,E2 -17461.46} C_VEL
LIN {X 0,Y 276.057,Z 472.856,A -85,B 0,C 180,E1 -17463.649,E2 -17463.649} C_VEL
LIN {X 0,Y 276.441,Z 466.666,A -85,B 0,C 180,E1 -17465.471,E2 -17465.471} C_VEL
LIN {X 0,Y 276.693,Z 458.845,A -85,B 0,C 180,E1 -17467.296,E2 -17467.296} C_VEL
LIN {X 0,Y 277.132,Z 450.015,A -85,B 0,C 180,E1 -17468.936,E2 -17468.936} C_VEL
LIN {X 0,Y 277.572,Z 440.07,A -85,B 0,C 180,E1 -17470.393,E2 -17470.393} C_VEL
LIN {X 0,Y 277.816,Z 432.379,A -85,B 0,C 180,E1 -17471.306,E2 -17471.306} C_VEL
LIN {X 0,Y 276.626,Z 421.264,A -85,B 0,C 180,E1 -17472.378,E2 -17472.378} C_VEL
LIN {X 0,Y 276.061,Z 414.346,A -85,B 0,C 180,E1 -17472.918,E2 -17472.918} C_VEL
LIN {X 0,Y 276.274,Z 408.049,A -85,B 0,C 180,E1 -17477.01,E2 -17477.01} C_VEL
LIN {X 0,Y 276.625,Z 402.276,A -85,B 0,C 180,E1 -17480.836,E2 -17480.836} C_VEL
LIN {X 0,Y 277.007,Z 396.503,A -85,B 0,C 180,E1 -17484.747,E2 -17484.747} C_VEL
LIN {X 0,Y 277.494,Z 390.668,A -85,B 0,C 180,E1 -17488.765,E2 -17488.765} C_VEL
LIN {X 0,Y 277.723,Z 387.082,A -85,B 0,C 180,E1 -17491.293,E2 -17491.293} C_VEL
LIN {X 0,Y 277.494,Z 385.918,A -85,B 0,C 180,E1 -17492.321,E2 -17492.321} C_VEL
LIN {X 0,Y 277.301,Z 385.94,A -85,B 0,C 180,E1 -17495.804,E2 -17495.804} C_VEL
LIN {X 0,Y 277.236,Z 385.95,A -85,B 0,C 180,E1 -17499.328,E2 -17499.328} C_VEL
LIN {X 0,Y 277.219,Z 385.951,A -85,B 0,C 180,E1 -17503.197,E2 -17503.197} C_VEL
LIN {X 0,Y 277.221,Z 385.951,A -85,B 0,C 180,E1 -17507.324,E2 -17507.324} C_VEL
LIN {X 0,Y 277.264,Z 385.944,A -85,B 0,C 180,E1 -17511.793,E2 -17511.793} C_VEL
LIN {X 0,Y 277.286,Z 385.945,A -85,B 0,C 180,E1 -17514.341,E2 -17514.341} C_VEL
LIN {X 0,Y 277.246,Z 385.948,A -85,B 0,C 180,E1 -17517.836,E2 -17517.836} C_VEL
LIN {X 0,Y 277.271,Z 385.944,A -85,B 0,C 180,E1 -17521.21,E2 -17521.21} C_VEL
LIN {X 0,Y 277.316,Z 385.943,A -85,B 0,C 180,E1 -17524.479,E2 -17524.479} C_VEL
LIN {X 0,Y 277.294,Z 385.941,A -85,B 0,C 180,E1 -17527.655,E2 -17527.655} C_VEL
LIN {X 0,Y 277.348,Z 385.936,A -85,B 0,C 180,E1 -17530.766,E2 -17530.766} C_VEL
LIN {X 0,Y 277.438,Z 385.923,A -85,B 0,C 180,E1 -17535.326,E2 -17535.326} C_VEL
LIN {X 0,Y 277.464,Z 385.922,A -85,B 0,C 180,E1 -17539.787,E2 -17539.787} C_VEL
LIN {X 0,Y 277.644,Z 385.898,A -85,B 0,C 180,E1 -17542.729,E2 -17542.729} C_VEL
LIN {X 0,Y 277.824,Z 385.877,A -85,B 0,C 180,E1 -17548.55,E2 -17548.55} C_VEL
LIN {X 0,Y 277.825,Z 385.876,A -85,B 0,C 180,E1 -17551.449,E2 -17551.449} C_VEL
LIN {X 0,Y 277.652,Z 385.897,A -85,B 0,C 180,E1 -17557.271,E2 -17557.271} C_VEL
LIN {X 0,Y 277.51,Z 385.916,A -85,B 0,C 180,E1 -17560.211,E2 -17560.211} C_VEL
LIN {X 0,Y 277.438,Z 385.923,A -85,B 0,C 180,E1 -17564.674,E2 -17564.674} C_VEL
LIN {X 0,Y 277.35,Z 385.936,A -85,B 0,C 180,E1 -17569.233,E2 -17569.233} C_VEL
LIN {X 0,Y 277.332,Z 385.939,A -85,B 0,C 180,E1 -17573.92,E2 -17573.92} C_VEL
LIN {X 0,Y 277.326,Z 385.942,A -85,B 0,C 180,E1 -17577.504,E2 -17577.504} C_VEL
LIN {X 0,Y 277.274,Z 385.943,A -85,B 0,C 180,E1 -17580.481,E2 -17580.481} C_VEL
LIN {X 0,Y 277.256,Z 385.948,A -85,B 0,C 180,E1 -17583.894,E2 -17583.894} C_VEL
LIN {X 0,Y 277.284,Z 385.945,A -85,B 0,C 180,E1 -17587.467,E2 -17587.467} C_VEL
LIN {X 0,Y 277.212,Z 385.955,A -85,B 0,C 180,E1 -17591.236,E2 -17591.236} C_VEL
LIN {X 0,Y 277.202,Z 385.957,A -85,B 0,C 180,E1 -17595.226,E2 -17595.226} C_VEL
LIN {X 0,Y 277.224,Z 385.952,A -85,B 0,C 180,E1 -17599.512,E2 -17599.512} C_VEL
LIN {X 0,Y 277.266,Z 385.946,A -85,B 0,C 180,E1 -17602.53,E2 -17602.53} C_VEL
LIN {X 0,Y 277.248,Z 385.946,A -85,B 0,C 180,E1 -17606.104,E2 -17606.104} C_VEL
LIN {X 0,Y 277.263,Z 385.946,A -85,B 0,C 180,E1 -17609.538,E2 -17609.538} C_VEL
LIN {X 0,Y 277.361,Z 385.937,A -85,B 0,C 180,E1 -17612.864,E2 -17612.864} C_VEL
LIN {X 0,Y 277.331,Z 385.936,A -85,B 0,C 180,E1 -17616.079,E2 -17616.079} C_VEL
LIN {X 0,Y 277.347,Z 385.939,A -85,B 0,C 180,E1 -17620.766,E2 -17620.766} C_VEL
LIN {X 0,Y 277.437,Z 385.924,A -85,B 0,C 180,E1 -17625.326,E2 -17625.326} C_VEL
LIN {X 0,Y 277.509,Z 385.914,A -85,B 0,C 180,E1 -17629.789,E2 -17629.789} C_VEL
LIN {X 0,Y 277.655,Z 385.9,A -85,B 0,C 180,E1 -17632.729,E2 -17632.729} C_VEL
LIN {X 0,Y 277.823,Z 385.879,A -85,B 0,C 180,E1 -17638.55,E2 -17638.55} C_VEL
LIN {X 0,Y 277.826,Z 385.874,A -85,B 0,C 180,E1 -17641.449,E2 -17641.449} C_VEL
LIN {X 0,Y 277.655,Z 385.896,A -85,B 0,C 180,E1 -17647.271,E2 -17647.271} C_VEL
LIN {X 0,Y 277.508,Z 385.918,A -85,B 0,C 180,E1 -17650.211,E2 -17650.211} C_VEL
LIN {X 0,Y 277.436,Z 385.925,A -85,B 0,C 180,E1 -17654.674,E2 -17654.674} C_VEL
LIN {X 0,Y 277.347,Z 385.934,A -85,B 0,C 180,E1 -17659.234,E2 -17659.234} C_VEL
LIN {X 0,Y 277.321,Z 385.941,A -85,B 0,C 180,E1 -17664.17,E2 -17664.17} C_VEL
LIN {X 0,Y 277.312,Z 385.939,A -85,B 0,C 180,E1 -17665.458,E2 -17665.458} C_VEL
LIN {X 0,Y 276.681,Z 386.021,A -85,B 0,C 180,E1 -17666.671,E2 -17666.671} C_VEL
LIN {X 0,Y 273.8,Z 386.383,A -85,B 0,C 180,E1 -17668.644,E2 -17668.644} C_VEL
LIN {X 0,Y 271.323,Z 386.688,A -85,B 0,C 180,E1 -17670.248,E2 -17670.248} C_VEL
LIN {X 0,Y 270.253,Z 386.82,A -85,B 0,C 180,E1 -17671.493,E2 -17671.493} C_VEL
LIN {X 0,Y 270.164,Z 386.826,A -85,B 0,C 180,E1 -17671.915,E2 -17671.915} C_VEL
LIN {X 0,Y 270.216,Z 386.822,A -85,B 0,C 180,E1 -17674.903,E2 -17674.903} C_VEL
LIN {X 0,Y 270.223,Z 386.822,A -85,B 0,C 180,E1 -17678.717,E2 -17678.717} C_VEL
LIN {X 0,Y 270.173,Z 386.828,A -85,B 0,C 180,E1 -17683.251,E2 -17683.251} C_VEL
LIN {X 0,Y 270.26,Z 386.992,A -85,B 0,C 180,E1 -17687.857,E2 -17687.857} C_VEL
LIN {X 0,Y 272.167,Z 396.5,A -85,B 0,C 180,E1 -17692.464,E2 -17692.464} C_VEL
LIN {X 0,Y 274.45,Z 407.379,A -85,B 0,C 180,E1 -17697.469,E2 -17697.469} C_VEL
LIN {X 0,Y 274.936,Z 409.661,A -85,B 0,C 180,E1 -17698.48,E2 -17698.48} C_VEL
LIN {X 0,Y 275.018,Z 411.477,A -85,B 0,C 180,E1 -17699.263,E2 -17699.263} C_VEL
LIN {X 0,Y 272.552,Z 422.797,A -85,B 0,C 180,E1 -17704.001,E2 -17704.001} C_VEL
LIN {X 0,Y 270.419,Z 436.381,A -85,B 0,C 180,E1 -17709.706,E2 -17709.706} C_VEL
LIN {X 0,Y 270.23,Z 438.12,A -85,B 0,C 180,E1 -17710.437,E2 -17710.437} C_VEL
LIN {X 0,Y 270.517,Z 452.008,A -85,B 0,C 180,E1 -17711.246,E2 -17711.246} C_VEL
LIN {X 0,Y 271.361,Z 465.44,A -85,B 0,C 180,E1 -17712.364,E2 -17712.364} C_VEL
LIN {X 0,Y 271.889,Z 472.652,A -85,B 0,C 180,E1 -17713.123,E2 -17713.123} C_VEL
LIN {X 0,Y 271.175,Z 484.029,A -85,B 0,C 180,E1 -17714.595,E2 -17714.595} C_VEL
LIN {X 0,Y 270.392,Z 494.244,A -85,B 0,C 180,E1 -17716.28,E2 -17716.28} C_VEL
LIN {X 0,Y 269.848,Z 502.596,A -85,B 0,C 180,E1 -17717.974,E2 -17717.974} C_VEL
LIN {X 0,Y 269.484,Z 510.219,A -85,B 0,C 180,E1 -17719.861,E2 -17719.861} C_VEL
LIN {X 0,Y 269.351,Z 517.521,A -85,B 0,C 180,E1 -17722.127,E2 -17722.127} C_VEL
LIN {X 0,Y 269.382,Z 522.358,A -85,B 0,C 180,E1 -17724.01,E2 -17724.01} C_VEL
LIN {X 0,Y 269.432,Z 526.857,A -85,B 0,C 180,E1 -17726.261,E2 -17726.261} C_VEL
LIN {X 0,Y 269.403,Z 530.079,A -85,B 0,C 180,E1 -17728.505,E2 -17728.505} C_VEL
LIN {X 0,Y 269.325,Z 531.56,A -85,B 0,C 180,E1 -17730,E2 -17730} C_VEL
LIN {X 0,Y 269.235,Z 532.584,A -85,B 0,C 180,E1 -17731.496,E2 -17731.496} C_VEL
LIN {X 0,Y 268.938,Z 533.145,A -85,B 0,C 180,E1 -17732.996,E2 -17732.996} C_VEL
LIN {X 0,Y 268.585,Z 532.957,A -85,B 0,C 180,E1 -17736.008,E2 -17736.008} C_VEL
LIN {X 0,Y 268.568,Z 532.277,A -85,B 0,C 180,E1 -17737.518,E2 -17737.518} C_VEL
LIN {X 0,Y 268.911,Z 529.656,A -85,B 0,C 180,E1 -17740.542,E2 -17740.542} C_VEL
LIN {X 0,Y 269.717,Z 526.643,A -85,B 0,C 180,E1 -17742.796,E2 -17742.796} C_VEL
LIN {X 0,Y 271.122,Z 522.671,A -85,B 0,C 180,E1 -17745.024,E2 -17745.024} C_VEL
LIN {X 0,Y 272.809,Z 517.655,A -85,B 0,C 180,E1 -17747.233,E2 -17747.233} C_VEL
LIN {X 0,Y 275.543,Z 510.304,A -85,B 0,C 180,E1 -17749.753,E2 -17749.753} C_VEL
LIN {X 0,Y 278.491,Z 502.518,A -85,B 0,C 180,E1 -17751.854,E2 -17751.854} C_VEL
LIN {X 0,Y 282.006,Z 492.955,A -85,B 0,C 180,E1 -17753.89,E2 -17753.89} C_VEL
LIN {X 0,Y 284.344,Z 485.431,A -85,B 0,C 180,E1 -17755.237,E2 -17755.237} C_VEL
LIN {X 0,Y 286.096,Z 477.093,A -85,B 0,C 180,E1 -17756.632,E2 -17756.632} C_VEL
LIN {X 0,Y 286.759,Z 467.357,A -85,B 0,C 180,E1 -17758.236,E2 -17758.236} C_VEL
LIN {X 0,Y 286.375,Z 455.923,A -85,B 0,C 180,E1 -17760.14,E2 -17760.14} C_VEL
LIN {X 0,Y 285.193,Z 446.394,A -85,B 0,C 180,E1 -17761.787,E2 -17761.787} C_VEL
LIN {X 0,Y 283.495,Z 438.047,A -85,B 0,C 180,E1 -17763.353,E2 -17763.353} C_VEL
LIN {X 0,Y 281.548,Z 433.159,A -85,B 0,C 180,E1 -17764.652,E2 -17764.652} C_VEL
LIN {X 0,Y 281.052,Z 430.568,A -85,B 0,C 180,E1 -17766.881,E2 -17766.881} C_VEL
LIN {X 0,Y 280.331,Z 427.044,A -85,B 0,C 180,E1 -17770.68,E2 -17770.68} C_VEL
LIN {X 0,Y 279.904,Z 425.265,A -85,B 0,C 180,E1 -17773.268,E2 -17773.268} C_VEL
LIN {X 0,Y 279.622,Z 424.23,A -85,B 0,C 180,E1 -17775.271,E2 -17775.271} C_VEL
LIN {X 0,Y 279.352,Z 423.511,A -85,B 0,C 180,E1 -17777.213,E2 -17777.213} C_VEL
LIN {X 0,Y 278.829,Z 422.857,A -85,B 0,C 180,E1 -17781.386,E2 -17781.386} C_VEL
LIN {X 0,Y 278.474,Z 423.107,A -85,B 0,C 180,E1 -17784.517,E2 -17784.517} C_VEL
LIN {X 0,Y 277.809,Z 424.164,A -85,B 0,C 180,E1 -17787.91,E2 -17787.91} C_VEL
LIN {X 0,Y 277.459,Z 424.888,A -85,B 0,C 180,E1 -17789.183,E2 -17789.183} C_VEL
LIN {X 0,Y 279.081,Z 428.736,A -85,B 0,C 180,E1 -17790.698,E2 -17790.698} C_VEL
LIN {X 0,Y 279.943,Z 430.921,A -85,B 0,C 180,E1 -17791.51,E2 -17791.51} C_VEL
LIN {X 0,Y 282.642,Z 438.374,A -85,B 0,C 180,E1 -17794.032,E2 -17794.032} C_VEL
LIN {X 0,Y 284.691,Z 446.373,A -85,B 0,C 180,E1 -17796.417,E2 -17796.417} C_VEL
LIN {X 0,Y 285.765,Z 453.265,A -85,B 0,C 180,E1 -17798.352,E2 -17798.352} C_VEL
LIN {X 0,Y 286.002,Z 460.681,A -85,B 0,C 180,E1 -17800.425,E2 -17800.425} C_VEL
LIN {X 0,Y 285.859,Z 462.375,A -85,B 0,C 180,E1 -17800.888,E2 -17800.888} C_VEL
LIN {X 0,Y 283.113,Z 469.561,A -85,B 0,C 180,E1 -17802.669,E2 -17802.669} C_VEL
LIN {X 0,Y 279.981,Z 476.102,A -85,B 0,C 180,E1 -17804.718,E2 -17804.718} C_VEL
LIN {X 0,Y 277.28,Z 481.015,A -85,B 0,C 180,E1 -17806.814,E2 -17806.814} C_VEL
LIN {X 0,Y 275.713,Z 483.447,A -85,B 0,C 180,E1 -17808.234,E2 -17808.234} C_VEL
LIN {X 0,Y 274.233,Z 485.283,A -85,B 0,C 180,E1 -17809.666,E2 -17809.666} C_VEL
LIN {X 0,Y 272.888,Z 486.546,A -85,B 0,C 180,E1 -17811.111,E2 -17811.111} C_VEL
LIN {X 0,Y 271.721,Z 487.22,A -85,B 0,C 180,E1 -17812.57,E2 -17812.57} C_VEL
LIN {X 0,Y 270.777,Z 487.305,A -85,B 0,C 180,E1 -17814.041,E2 -17814.041} C_VEL
LIN {X 0,Y 270.054,Z 486.776,A -85,B 0,C 180,E1 -17815.522,E2 -17815.522} C_VEL
LIN {X 0,Y 269.51,Z 485.642,A -85,B 0,C 180,E1 -17817.011,E2 -17817.011} C_VEL
LIN {X 0,Y 269.061,Z 482.795,A -85,B 0,C 180,E1 -17819.252,E2 -17819.252} C_VEL
LIN {X 0,Y 268.818,Z 478.491,A -85,B 0,C 180,E1 -17821.498,E2 -17821.498} C_VEL
LIN {X 0,Y 268.981,Z 472.533,A -85,B 0,C 180,E1 -17823.745,E2 -17823.745} C_VEL
LIN {X 0,Y 269.394,Z 466.068,A -85,B 0,C 180,E1 -17825.614,E2 -17825.614} C_VEL
LIN {X 0,Y 269.621,Z 457.876,A -85,B 0,C 180,E1 -17827.489,E2 -17827.489} C_VEL
LIN {X 0,Y 270.046,Z 448.62,A -85,B 0,C 180,E1 -17829.173,E2 -17829.173} C_VEL
LIN {X 0,Y 270.616,Z 438.276,A -85,B 0,C 180,E1 -17830.664,E2 -17830.664} C_VEL
LIN {X 0,Y 270.642,Z 431.896,A -85,B 0,C 180,E1 -17831.421,E2 -17831.421} C_VEL
LIN {X 0,Y 269.398,Z 420.518,A -85,B 0,C 180,E1 -17832.525,E2 -17832.525} C_VEL
LIN {X 0,Y 268.999,Z 414.597,A -85,B 0,C 180,E1 -17833.023,E2 -17833.023} C_VEL
LIN {X 0,Y 269.232,Z 407.895,A -85,B 0,C 180,E1 -17837.469,E2 -17837.469} C_VEL
LIN {X 0,Y 269.605,Z 402.083,A -85,B 0,C 180,E1 -17841.405,E2 -17841.405} C_VEL
LIN {X 0,Y 270.018,Z 396.26,A -85,B 0,C 180,E1 -17845.434,E2 -17845.434} C_VEL
LIN {X 0,Y 270.554,Z 390.374,A -85,B 0,C 180,E1 -17849.575,E2 -17849.575} C_VEL
LIN {X 0,Y 270.524,Z 387.097,A -85,B 0,C 180,E1 -17851.96,E2 -17851.96} C_VEL
LIN {X 0,Y 270.438,Z 386.797,A -85,B 0,C 180,E1 -17852.191,E2 -17852.191} C_VEL
LIN {X 0,Y 270.225,Z 386.825,A -85,B 0,C 180,E1 -17856.74,E2 -17856.74} C_VEL
LIN {X 0,Y 270.172,Z 386.831,A -85,B 0,C 180,E1 -17861.028,E2 -17861.028} C_VEL
LIN {X 0,Y 270.168,Z 386.83,A -85,B 0,C 180,E1 -17865.383,E2 -17865.383} C_VEL
LIN {X 0,Y 270.176,Z 386.828,A -85,B 0,C 180,E1 -17869.434,E2 -17869.434} C_VEL
LIN {X 0,Y 270.228,Z 386.821,A -85,B 0,C 180,E1 -17873.731,E2 -17873.731} C_VEL
LIN {X 0,Y 270.205,Z 386.826,A -85,B 0,C 180,E1 -17876.893,E2 -17876.893} C_VEL
LIN {X 0,Y 270.222,Z 386.825,A -85,B 0,C 180,E1 -17880.386,E2 -17880.386} C_VEL
LIN {X 0,Y 270.265,Z 386.818,A -85,B 0,C 180,E1 -17883.764,E2 -17883.764} C_VEL
LIN {X 0,Y 270.239,Z 386.82,A -85,B 0,C 180,E1 -17887.039,E2 -17887.039} C_VEL
LIN {X 0,Y 270.305,Z 386.815,A -85,B 0,C 180,E1 -17890.245,E2 -17890.245} C_VEL
LIN {X 0,Y 270.406,Z 386.799,A -85,B 0,C 180,E1 -17894.935,E2 -17894.935} C_VEL
LIN {X 0,Y 270.416,Z 386.798,A -85,B 0,C 180,E1 -17899.518,E2 -17899.518} C_VEL
LIN {X 0,Y 270.602,Z 386.777,A -85,B 0,C 180,E1 -17902.538,E2 -17902.538} C_VEL
LIN {X 0,Y 270.79,Z 386.753,A -85,B 0,C 180,E1 -17908.513,E2 -17908.513} C_VEL
LIN {X 0,Y 270.791,Z 386.753,A -85,B 0,C 180,E1 -17911.487,E2 -17911.487} C_VEL
LIN {X 0,Y 270.611,Z 386.775,A -85,B 0,C 180,E1 -17917.461,E2 -17917.461} C_VEL
LIN {X 0,Y 270.445,Z 386.795,A -85,B 0,C 180,E1 -17920.481,E2 -17920.481} C_VEL
LIN {X 0,Y 270.406,Z 386.799,A -85,B 0,C 180,E1 -17925.064,E2 -17925.064} C_VEL
LIN {X 0,Y 270.306,Z 386.815,A -85,B 0,C 180,E1 -17929.755,E2 -17929.755} C_VEL
LIN {X 0,Y 270.276,Z 386.816,A -85,B 0,C 180,E1 -17934.585,E2 -17934.585} C_VEL
LIN {X 0,Y 270.272,Z 386.817,A -85,B 0,C 180,E1 -17937.909,E2 -17937.909} C_VEL
LIN {X 0,Y 270.186,Z 386.829,A -85,B 0,C 180,E1 -17941.348,E2 -17941.348} C_VEL
LIN {X 0,Y 270.217,Z 386.824,A -85,B 0,C 180,E1 -17944.903,E2 -17944.903} C_VEL
LIN {X 0,Y 270.224,Z 386.821,A -85,B 0,C 180,E1 -17948.717,E2 -17948.717} C_VEL
LIN {X 0,Y 270.166,Z 386.834,A -85,B 0,C 180,E1 -17953.249,E2 -17953.249} C_VEL
LIN {X 0,Y 270.173,Z 386.83,A -85,B 0,C 180,E1 -17957.442,E2 -17957.442} C_VEL
LIN {X 0,Y 270.208,Z 386.827,A -85,B 0,C 180,E1 -17961.374,E2 -17961.374} C_VEL
LIN {X 0,Y 270.203,Z 386.828,A -85,B 0,C 180,E1 -17965.094,E2 -17965.094} C_VEL
LIN {X 0,Y 270.202,Z 386.829,A -85,B 0,C 180,E1 -17969.13,E2 -17969.13} C_VEL
LIN {X 0,Y 270.266,Z 386.817,A -85,B 0,C 180,E1 -17972.145,E2 -17972.145} C_VEL
LIN {X 0,Y 270.279,Z 386.815,A -85,B 0,C 180,E1 -17975.519,E2 -17975.519} C_VEL
LIN {X 0,Y 270.303,Z 386.813,A -85,B 0,C 180,E1 -17980.244,E2 -17980.244} C_VEL
LIN {X 0,Y 270.405,Z 386.803,A -85,B 0,C 180,E1 -17984.935,E2 -17984.935} C_VEL
LIN {X 0,Y 270.444,Z 386.794,A -85,B 0,C 180,E1 -17989.519,E2 -17989.519} C_VEL
LIN {X 0,Y 270.613,Z 386.776,A -85,B 0,C 180,E1 -17992.539,E2 -17992.539} C_VEL
LIN {X 0,Y 270.789,Z 386.755,A -85,B 0,C 180,E1 -17998.513,E2 -17998.513} C_VEL
LIN {X 0,Y 270.792,Z 386.751,A -85,B 0,C 180,E1 -18001.487,E2 -18001.487} C_VEL
LIN {X 0,Y 270.613,Z 386.773,A -85,B 0,C 180,E1 -18007.461,E2 -18007.461} C_VEL
LIN {X 0,Y 270.443,Z 386.798,A -85,B 0,C 180,E1 -18010.481,E2 -18010.481} C_VEL
LIN {X 0,Y 270.404,Z 386.799,A -85,B 0,C 180,E1 -18015.064,E2 -18015.064} C_VEL
LIN {X 0,Y 270.303,Z 386.814,A -85,B 0,C 180,E1 -18019.755,E2 -18019.755} C_VEL
LIN {X 0,Y 270.275,Z 386.816,A -85,B 0,C 180,E1 -18024.585,E2 -18024.585} C_VEL
LIN {X 0,Y 270.271,Z 386.819,A -85,B 0,C 180,E1 -18027.909,E2 -18027.909} C_VEL
LIN {X 0,Y 270.164,Z 386.826,A -85,B 0,C 180,E1 -18031.915,E2 -18031.915} C_VEL
LIN {X 0,Y 269.497,Z 386.913,A -85,B 0,C 180,E1 -18033.161,E2 -18033.161} C_VEL
LIN {X 0,Y 266.668,Z 387.264,A -85,B 0,C 180,E1 -18035.191,E2 -18035.191} C_VEL
LIN {X 0,Y 264.263,Z 387.567,A -85,B 0,C 180,E1 -18036.842,E2 -18036.842} C_VEL
LIN {X 0,Y 263.223,Z 387.697,A -85,B 0,C 180,E1 -18038.12,E2 -18038.12} C_VEL
LIN {X 0,Y 263.134,Z 387.706,A -85,B 0,C 180,E1 -18038.554,E2 -18038.554} C_VEL
LIN {X 0,Y 263.126,Z 387.708,A -85,B 0,C 180,E1 -18041.893,E2 -18041.893} C_VEL
LIN {X 0,Y 263.136,Z 387.709,A -85,B 0,C 180,E1 -18046.148,E2 -18046.148} C_VEL
LIN {X 0,Y 263.227,Z 387.85,A -85,B 0,C 180,E1 -18047.542,E2 -18047.542} C_VEL
LIN {X 0,Y 265.163,Z 397.686,A -85,B 0,C 180,E1 -18052.439,E2 -18052.439} C_VEL
LIN {X 0,Y 267.332,Z 407.868,A -85,B 0,C 180,E1 -18057.274,E2 -18057.274} C_VEL
LIN {X 0,Y 267.838,Z 410.207,A -85,B 0,C 180,E1 -18058.346,E2 -18058.346} C_VEL
LIN {X 0,Y 267.911,Z 412.199,A -85,B 0,C 180,E1 -18059.234,E2 -18059.234} C_VEL
LIN {X 0,Y 265.321,Z 423.777,A -85,B 0,C 180,E1 -18064.239,E2 -18064.239} C_VEL
LIN {X 0,Y 263.17,Z 437.816,A -85,B 0,C 180,E1 -18070.347,E2 -18070.347} C_VEL
LIN {X 0,Y 263.348,Z 450.664,A -85,B 0,C 180,E1 -18071.12,E2 -18071.12} C_VEL
LIN {X 0,Y 264.141,Z 463.426,A -85,B 0,C 180,E1 -18072.184,E2 -18072.184} C_VEL
LIN {X 0,Y 264.774,Z 473.086,A -85,B 0,C 180,E1 -18073.222,E2 -18073.222} C_VEL
LIN {X 0,Y 264.041,Z 484.363,A -85,B 0,C 180,E1 -18074.761,E2 -18074.761} C_VEL
LIN {X 0,Y 263.299,Z 494.385,A -85,B 0,C 180,E1 -18076.494,E2 -18076.494} C_VEL
LIN {X 0,Y 262.758,Z 503.391,A -85,B 0,C 180,E1 -18078.428,E2 -18078.428} C_VEL
LIN {X 0,Y 262.382,Z 511.997,A -85,B 0,C 180,E1 -18080.752,E2 -18080.752} C_VEL
LIN {X 0,Y 262.37,Z 518.379,A -85,B 0,C 180,E1 -18082.931,E2 -18082.931} C_VEL
LIN {X 0,Y 262.411,Z 523.935,A -85,B 0,C 180,E1 -18085.392,E2 -18085.392} C_VEL
LIN {X 0,Y 262.436,Z 527.768,A -85,B 0,C 180,E1 -18087.698,E2 -18087.698} C_VEL
LIN {X 0,Y 262.32,Z 530.384,A -85,B 0,C 180,E1 -18090,E2 -18090} C_VEL
LIN {X 0,Y 262.205,Z 531.503,A -85,B 0,C 180,E1 -18091.536,E2 -18091.536} C_VEL
LIN {X 0,Y 261.892,Z 532.148,A -85,B 0,C 180,E1 -18093.077,E2 -18093.077} C_VEL
LIN {X 0,Y 261.603,Z 532.388,A -85,B 0,C 180,E1 -18094.623,E2 -18094.623} C_VEL
LIN {X 0,Y 261.51,Z 532.202,A -85,B 0,C 180,E1 -18096.171,E2 -18096.171} C_VEL
LIN {X 0,Y 261.631,Z 530.639,A -85,B 0,C 180,E1 -18099.275,E2 -18099.275} C_VEL
LIN {X 0,Y 261.89,Z 529.265,A -85,B 0,C 180,E1 -18100.827,E2 -18100.827} C_VEL
LIN {X 0,Y 262.768,Z 526.459,A -85,B 0,C 180,E1 -18103.141,E2 -18103.141} C_VEL
LIN {X 0,Y 264.737,Z 521.238,A -85,B 0,C 180,E1 -18106.185,E2 -18106.185} C_VEL
LIN {X 0,Y 267.084,Z 515.45,A -85,B 0,C 180,E1 -18108.684,E2 -18108.684} C_VEL
LIN {X 0,Y 269.968,Z 508.639,A -85,B 0,C 180,E1 -18110.975,E2 -18110.975} C_VEL
LIN {X 0,Y 273.127,Z 500.76,A -85,B 0,C 180,E1 -18113.105,E2 -18113.105} C_VEL
LIN {X 0,Y 276.974,Z 491.116,A -85,B 0,C 180,E1 -18115.152,E2 -18115.152} C_VEL
LIN {X 0,Y 279.746,Z 481.613,A -85,B 0,C 180,E1 -18116.886,E2 -18116.886} C_VEL
LIN {X 0,Y 281.122,Z 471.471,A -85,B 0,C 180,E1 -18118.687,E2 -18118.687} C_VEL
LIN {X 0,Y 281.324,Z 461.618,A -85,B 0,C 180,E1 -18120.435,E2 -18120.435} C_VEL
LIN {X 0,Y 280.66,Z 450.971,A -85,B 0,C 180,E1 -18122.4,E2 -18122.4} C_VEL
LIN {X 0,Y 279.551,Z 443.262,A -85,B 0,C 180,E1 -18123.939,E2 -18123.939} C_VEL
LIN {X 0,Y 277.957,Z 438.836,A -85,B 0,C 180,E1 -18125.16,E2 -18125.16} C_VEL
LIN {X 0,Y 274.61,Z 433.238,A -85,B 0,C 180,E1 -18127.498,E2 -18127.498} C_VEL
LIN {X 0,Y 274.192,Z 432.04,A -85,B 0,C 180,E1 -18127.964,E2 -18127.964} C_VEL
LIN {X 0,Y 273.848,Z 430.281,A -85,B 0,C 180,E1 -18129.911,E2 -18129.911} C_VEL
LIN {X 0,Y 273.512,Z 428.754,A -85,B 0,C 180,E1 -18131.919,E2 -18131.919} C_VEL
LIN {X 0,Y 273.192,Z 427.49,A -85,B 0,C 180,E1 -18133.995,E2 -18133.995} C_VEL
LIN {X 0,Y 272.886,Z 426.503,A -85,B 0,C 180,E1 -18136.147,E2 -18136.147} C_VEL
LIN {X 0,Y 272.366,Z 425.589,A -85,B 0,C 180,E1 -18139.828,E2 -18139.828} C_VEL
LIN {X 0,Y 271.956,Z 425.523,A -85,B 0,C 180,E1 -18143.532,E2 -18143.532} C_VEL
LIN {X 0,Y 271.58,Z 426.09,A -85,B 0,C 180,E1 -18146.004,E2 -18146.004} C_VEL
LIN {X 0,Y 273.231,Z 429.776,A -85,B 0,C 180,E1 -18148.084,E2 -18148.084} C_VEL
LIN {X 0,Y 273.964,Z 430.68,A -85,B 0,C 180,E1 -18148.703,E2 -18148.703} C_VEL
LIN {X 0,Y 275.947,Z 436.339,A -85,B 0,C 180,E1 -18151.059,E2 -18151.059} C_VEL
LIN {X 0,Y 278.241,Z 444.338,A -85,B 0,C 180,E1 -18153.922,E2 -18153.922} C_VEL
LIN {X 0,Y 279.691,Z 451.739,A -85,B 0,C 180,E1 -18156.294,E2 -18156.294} C_VEL
LIN {X 0,Y 280.225,Z 459.391,A -85,B 0,C 180,E1 -18158.618,E2 -18158.618} C_VEL
LIN {X 0,Y 279.934,Z 464.742,A -85,B 0,C 180,E1 -18160.247,E2 -18160.247} C_VEL
LIN {X 0,Y 276.668,Z 472.287,A -85,B 0,C 180,E1 -18162.252,E2 -18162.252} C_VEL
LIN {X 0,Y 273.406,Z 478.342,A -85,B 0,C 180,E1 -18164.341,E2 -18164.341} C_VEL
LIN {X 0,Y 270.568,Z 482.823,A -85,B 0,C 180,E1 -18166.481,E2 -18166.481} C_VEL
LIN {X 0,Y 268.939,Z 485.034,A -85,B 0,C 180,E1 -18167.933,E2 -18167.933} C_VEL
LIN {X 0,Y 267.396,Z 486.662,A -85,B 0,C 180,E1 -18169.398,E2 -18169.398} C_VEL
LIN {X 0,Y 265.968,Z 487.722,A -85,B 0,C 180,E1 -18170.878,E2 -18170.878} C_VEL
LIN {X 0,Y 264.748,Z 488.193,A -85,B 0,C 180,E1 -18172.373,E2 -18172.373} C_VEL
LIN {X 0,Y 263.775,Z 488.07,A -85,B 0,C 180,E1 -18173.882,E2 -18173.882} C_VEL
LIN {X 0,Y 263.008,Z 487.361,A -85,B 0,C 180,E1 -18175.402,E2 -18175.402} C_VEL
LIN {X 0,Y 262.455,Z 486.062,A -85,B 0,C 180,E1 -18176.93,E2 -18176.93} C_VEL
LIN {X 0,Y 261.975,Z 482.949,A -85,B 0,C 180,E1 -18179.232,E2 -18179.232} C_VEL
LIN {X 0,Y 261.724,Z 478.339,A -85,B 0,C 180,E1 -18181.539,E2 -18181.539} C_VEL
LIN {X 0,Y 261.908,Z 472.077,A -85,B 0,C 180,E1 -18183.847,E2 -18183.847} C_VEL
LIN {X 0,Y 262.344,Z 465.363,A -85,B 0,C 180,E1 -18185.766,E2 -18185.766} C_VEL
LIN {X 0,Y 262.577,Z 456.831,A -85,B 0,C 180,E1 -18187.691,E2 -18187.691} C_VEL
LIN {X 0,Y 263.036,Z 447.145,A -85,B 0,C 180,E1 -18189.419,E2 -18189.419} C_VEL
LIN {X 0,Y 263.571,Z 436.187,A -85,B 0,C 180,E1 -18190.952,E2 -18190.952} C_VEL
LIN {X 0,Y 263.428,Z 431.149,A -85,B 0,C 180,E1 -18191.543,E2 -18191.543} C_VEL
LIN {X 0,Y 262.202,Z 419.32,A -85,B 0,C 180,E1 -18192.677,E2 -18192.677} C_VEL
LIN {X 0,Y 261.903,Z 414.974,A -85,B 0,C 180,E1 -18193.037,E2 -18193.037} C_VEL
LIN {X 0,Y 262.141,Z 408.881,A -85,B 0,C 180,E1 -18197.152,E2 -18197.152} C_VEL
LIN {X 0,Y 262.515,Z 403.029,A -85,B 0,C 180,E1 -18201.187,E2 -18201.187} C_VEL
LIN {X 0,Y 262.933,Z 397.161,A -85,B 0,C 180,E1 -18205.32,E2 -18205.32} C_VEL
LIN {X 0,Y 263.501,Z 391.252,A -85,B 0,C 180,E1 -18209.566,E2 -18209.566} C_VEL
LIN {X 0,Y 263.483,Z 387.958,A -85,B 0,C 180,E1 -18212.01,E2 -18212.01} C_VEL
LIN {X 0,Y 263.385,Z 387.673,A -85,B 0,C 180,E1 -18212.254,E2 -18212.254} C_VEL
LIN {X 0,Y 263.191,Z 387.701,A -85,B 0,C 180,E1 -18216.765,E2 -18216.765} C_VEL
LIN {X 0,Y 263.127,Z 387.705,A -85,B 0,C 180,E1 -18221.594,E2 -18221.594} C_VEL
LIN {X 0,Y 263.13,Z 387.706,A -85,B 0,C 180,E1 -18226.017,E2 -18226.017} C_VEL
LIN {X 0,Y 263.108,Z 387.709,A -85,B 0,C 180,E1 -18230.128,E2 -18230.128} C_VEL
LIN {X 0,Y 263.165,Z 387.702,A -85,B 0,C 180,E1 -18234.018,E2 -18234.018} C_VEL
LIN {X 0,Y 263.135,Z 387.705,A -85,B 0,C 180,E1 -18237.712,E2 -18237.712} C_VEL
LIN {X 0,Y 263.201,Z 387.697,A -85,B 0,C 180,E1 -18241.784,E2 -18241.784} C_VEL
LIN {X 0,Y 263.229,Z 387.694,A -85,B 0,C 180,E1 -18245.2,E2 -18245.2} C_VEL
LIN {X 0,Y 263.267,Z 387.688,A -85,B 0,C 180,E1 -18249.694,E2 -18249.694} C_VEL
LIN {X 0,Y 263.354,Z 387.68,A -85,B 0,C 180,E1 -18254.522,E2 -18254.522} C_VEL
LIN {X 0,Y 263.358,Z 387.677,A -85,B 0,C 180,E1 -18259.234,E2 -18259.234} C_VEL
LIN {X 0,Y 263.561,Z 387.655,A -85,B 0,C 180,E1 -18262.338,E2 -18262.338} C_VEL
LIN {X 0,Y 263.754,Z 387.63,A -85,B 0,C 180,E1 -18268.473,E2 -18268.473} C_VEL
LIN {X 0,Y 263.755,Z 387.629,A -85,B 0,C 180,E1 -18271.527,E2 -18271.527} C_VEL
LIN {X 0,Y 263.573,Z 387.653,A -85,B 0,C 180,E1 -18277.661,E2 -18277.661} C_VEL
LIN {X 0,Y 263.377,Z 387.675,A -85,B 0,C 180,E1 -18280.765,E2 -18280.765} C_VEL
LIN {X 0,Y 263.354,Z 387.68,A -85,B 0,C 180,E1 -18285.478,E2 -18285.478} C_VEL
LIN {X 0,Y 263.272,Z 387.687,A -85,B 0,C 180,E1 -18290.306,E2 -18290.306} C_VEL
LIN {X 0,Y 263.211,Z 387.698,A -85,B 0,C 180,E1 -18295.291,E2 -18295.291} C_VEL
LIN {X 0,Y 263.177,Z 387.699,A -85,B 0,C 180,E1 -18298.73,E2 -18298.73} C_VEL
LIN {X 0,Y 263.135,Z 387.705,A -85,B 0,C 180,E1 -18302.288,E2 -18302.288} C_VEL
LIN {X 0,Y 263.19,Z 387.699,A -85,B 0,C 180,E1 -18305.978,E2 -18305.978} C_VEL
LIN {X 0,Y 263.117,Z 387.708,A -85,B 0,C 180,E1 -18309.87,E2 -18309.87} C_VEL
LIN {X 0,Y 263.105,Z 387.709,A -85,B 0,C 180,E1 -18313.988,E2 -18313.988} C_VEL
LIN {X 0,Y 263.126,Z 387.705,A -85,B 0,C 180,E1 -18318.406,E2 -18318.406} C_VEL
LIN {X 0,Y 263.183,Z 387.702,A -85,B 0,C 180,E1 -18323.237,E2 -18323.237} C_VEL
LIN {X 0,Y 263.135,Z 387.705,A -85,B 0,C 180,E1 -18327.712,E2 -18327.712} C_VEL
LIN {X 0,Y 263.203,Z 387.697,A -85,B 0,C 180,E1 -18331.783,E2 -18331.783} C_VEL
LIN {X 0,Y 263.228,Z 387.695,A -85,B 0,C 180,E1 -18335.2,E2 -18335.2} C_VEL
LIN {X 0,Y 263.265,Z 387.689,A -85,B 0,C 180,E1 -18339.693,E2 -18339.693} C_VEL
LIN {X 0,Y 263.353,Z 387.68,A -85,B 0,C 180,E1 -18344.522,E2 -18344.522} C_VEL
LIN {X 0,Y 263.377,Z 387.675,A -85,B 0,C 180,E1 -18349.234,E2 -18349.234} C_VEL
LIN {X 0,Y 263.575,Z 387.651,A -85,B 0,C 180,E1 -18352.338,E2 -18352.338} C_VEL
LIN {X 0,Y 263.753,Z 387.632,A -85,B 0,C 180,E1 -18358.473,E2 -18358.473} C_VEL
LIN {X 0,Y 263.756,Z 387.627,A -85,B 0,C 180,E1 -18361.527,E2 -18361.527} C_VEL
LIN {X 0,Y 263.575,Z 387.65,A -85,B 0,C 180,E1 -18367.661,E2 -18367.661} C_VEL
LIN {X 0,Y 263.376,Z 387.677,A -85,B 0,C 180,E1 -18370.765,E2 -18370.765} C_VEL
LIN {X 0,Y 263.353,Z 387.678,A -85,B 0,C 180,E1 -18375.478,E2 -18375.478} C_VEL
LIN {X 0,Y 263.265,Z 387.693,A -85,B 0,C 180,E1 -18380.306,E2 -18380.306} C_VEL
LIN {X 0,Y 263.21,Z 387.695,A -85,B 0,C 180,E1 -18385.291,E2 -18385.291} C_VEL
LIN {X 0,Y 263.167,Z 387.702,A -85,B 0,C 180,E1 -18388.731,E2 -18388.731} C_VEL
LIN {X 0,Y 263.134,Z 387.707,A -85,B 0,C 180,E1 -18392.288,E2 -18392.288} C_VEL
LIN {X 0,Y 263.189,Z 387.702,A -85,B 0,C 180,E1 -18395.978,E2 -18395.978} C_VEL
LIN {X 0,Y 263.134,Z 387.706,A -85,B 0,C 180,E1 -18398.554,E2 -18398.554} C_VEL
LIN {X 0,Y 262.444,Z 387.796,A -85,B 0,C 180,E1 -18399.831,E2 -18399.831} C_VEL
LIN {X 0,Y 259.562,Z 388.152,A -85,B 0,C 180,E1 -18401.913,E2 -18401.913} C_VEL
LIN {X 0,Y 257.142,Z 388.453,A -85,B 0,C 180,E1 -18403.607,E2 -18403.607} C_VEL
LIN {X 0,Y 256.13,Z 388.577,A -85,B 0,C 180,E1 -18404.92,E2 -18404.92} C_VEL
LIN {X 0,Y 256.061,Z 388.587,A -85,B 0,C 180,E1 -18405.365,E2 -18405.365} C_VEL
LIN {X 0,Y 256.143,Z 388.603,A -85,B 0,C 180,E1 -18407.169,E2 -18407.169} C_VEL
LIN {X 0,Y 257.875,Z 397.452,A -85,B 0,C 180,E1 -18411.74,E2 -18411.74} C_VEL
LIN {X 0,Y 259.765,Z 406.47,A -85,B 0,C 180,E1 -18416.182,E2 -18416.182} C_VEL
LIN {X 0,Y 260.763,Z 410.915,A -85,B 0,C 180,E1 -18418.294,E2 -18418.294} C_VEL
LIN {X 0,Y 260.516,Z 413.968,A -85,B 0,C 180,E1 -18419.686,E2 -18419.686} C_VEL
LIN {X 0,Y 257.878,Z 425.863,A -85,B 0,C 180,E1 -18425.012,E2 -18425.012} C_VEL
LIN {X 0,Y 256.062,Z 437.581,A -85,B 0,C 180,E1 -18430.301,E2 -18430.301} C_VEL
LIN {X 0,Y 256.237,Z 450.515,A -85,B 0,C 180,E1 -18431.096,E2 -18431.096} C_VEL
LIN {X 0,Y 257.012,Z 463.113,A -85,B 0,C 180,E1 -18432.186,E2 -18432.186} C_VEL
LIN {X 0,Y 257.682,Z 472.154,A -85,B 0,C 180,E1 -18433.185,E2 -18433.185} C_VEL
LIN {X 0,Y 257.026,Z 483.349,A -85,B 0,C 180,E1 -18434.741,E2 -18434.741} C_VEL
LIN {X 0,Y 256.217,Z 494.428,A -85,B 0,C 180,E1 -18436.719,E2 -18436.719} C_VEL
LIN {X 0,Y 255.751,Z 502.467,A -85,B 0,C 180,E1 -18438.508,E2 -18438.508} C_VEL
LIN {X 0,Y 255.374,Z 511.073,A -85,B 0,C 180,E1 -18440.895,E2 -18440.895} C_VEL
LIN {X 0,Y 255.385,Z 517.72,A -85,B 0,C 180,E1 -18443.23,E2 -18443.23} C_VEL
LIN {X 0,Y 255.421,Z 522.284,A -85,B 0,C 180,E1 -18445.265,E2 -18445.265} C_VEL
LIN {X 0,Y 255.462,Z 526.325,A -85,B 0,C 180,E1 -18447.635,E2 -18447.635} C_VEL
LIN {X 0,Y 255.329,Z 529.115,A -85,B 0,C 180,E1 -18450,E2 -18450} C_VEL
LIN {X 0,Y 255.181,Z 530.374,A -85,B 0,C 180,E1 -18451.578,E2 -18451.578} C_VEL
LIN {X 0,Y 254.864,Z 531.134,A -85,B 0,C 180,E1 -18453.162,E2 -18453.162} C_VEL
LIN {X 0,Y 254.441,Z 531.401,A -85,B 0,C 180,E1 -18456.343,E2 -18456.343} C_VEL
LIN {X 0,Y 254.442,Z 530.944,A -85,B 0,C 180,E1 -18457.938,E2 -18457.938} C_VEL
LIN {X 0,Y 254.886,Z 528.821,A -85,B 0,C 180,E1 -18461.129,E2 -18461.129} C_VEL
LIN {X 0,Y 255.835,Z 526.224,A -85,B 0,C 180,E1 -18463.504,E2 -18463.504} C_VEL
LIN {X 0,Y 257.337,Z 522.711,A -85,B 0,C 180,E1 -18465.849,E2 -18465.849} C_VEL
LIN {X 0,Y 259.615,Z 517.549,A -85,B 0,C 180,E1 -18468.469,E2 -18468.469} C_VEL
LIN {X 0,Y 262.843,Z 510.526,A -85,B 0,C 180,E1 -18471.16,E2 -18471.16} C_VEL
LIN {X 0,Y 266.128,Z 503.34,A -85,B 0,C 180,E1 -18473.336,E2 -18473.336} C_VEL
LIN {X 0,Y 270.035,Z 494.482,A -85,B 0,C 180,E1 -18475.432,E2 -18475.432} C_VEL
LIN {X 0,Y 273.18,Z 485.794,A -85,B 0,C 180,E1 -18477.171,E2 -18477.171} C_VEL
LIN {X 0,Y 274.892,Z 478.389,A -85,B 0,C 180,E1 -18478.589,E2 -18478.589} C_VEL
LIN {X 0,Y 275.975,Z 468.833,A -85,B 0,C 180,E1 -18480.404,E2 -18480.404} C_VEL
LIN {X 0,Y 276.127,Z 459.027,A -85,B 0,C 180,E1 -18482.31,E2 -18482.31} C_VEL
LIN {X 0,Y 275.632,Z 450.202,A -85,B 0,C 180,E1 -18484.122,E2 -18484.122} C_VEL
LIN {X 0,Y 275.392,Z 448.374,A -85,B 0,C 180,E1 -18484.524,E2 -18484.524} C_VEL
LIN {X 0,Y 274.328,Z 444.637,A -85,B 0,C 180,E1 -18485.616,E2 -18485.616} C_VEL
LIN {X 0,Y 270.896,Z 437.966,A -85,B 0,C 180,E1 -18488.51,E2 -18488.51} C_VEL
LIN {X 0,Y 267.315,Z 432.028,A -85,B 0,C 180,E1 -18492.595,E2 -18492.595} C_VEL
LIN {X 0,Y 266.534,Z 429.961,A -85,B 0,C 180,E1 -18494.343,E2 -18494.343} C_VEL
LIN {X 0,Y 266.043,Z 428.667,A -85,B 0,C 180,E1 -18497.704,E2 -18497.704} C_VEL
LIN {X 0,Y 265.816,Z 428.277,A -85,B 0,C 180,E1 -18499.533,E2 -18499.533} C_VEL
LIN {X 0,Y 266.437,Z 429.755,A -85,B 0,C 180,E1 -18502.311,E2 -18502.311} C_VEL
LIN {X 0,Y 268.537,Z 432.548,A -85,B 0,C 180,E1 -18505.803,E2 -18505.803} C_VEL
LIN {X 0,Y 270.665,Z 438.055,A -85,B 0,C 180,E1 -18508.967,E2 -18508.967} C_VEL
LIN {X 0,Y 272.259,Z 443.491,A -85,B 0,C 180,E1 -18511.362,E2 -18511.362} C_VEL
LIN {X 0,Y 273.771,Z 450.889,A -85,B 0,C 180,E1 -18514.125,E2 -18514.125} C_VEL
LIN {X 0,Y 274.503,Z 458.24,A -85,B 0,C 180,E1 -18516.62,E2 -18516.62} C_VEL
LIN {X 0,Y 274.29,Z 465.368,A -85,B 0,C 180,E1 -18518.979,E2 -18518.979} C_VEL
LIN {X 0,Y 273.905,Z 467.713,A -85,B 0,C 180,E1 -18519.733,E2 -18519.733} C_VEL
LIN {X 0,Y 270.237,Z 474.909,A -85,B 0,C 180,E1 -18521.815,E2 -18521.815} C_VEL
LIN {X 0,Y 266.851,Z 480.513,A -85,B 0,C 180,E1 -18523.946,E2 -18523.946} C_VEL
LIN {X 0,Y 263.879,Z 484.611,A -85,B 0,C 180,E1 -18526.131,E2 -18526.131} C_VEL
LIN {X 0,Y 262.163,Z 486.574,A -85,B 0,C 180,E1 -18527.616,E2 -18527.616} C_VEL
LIN {X 0,Y 260.557,Z 487.999,A -85,B 0,C 180,E1 -18529.117,E2 -18529.117} C_VEL
LIN {X 0,Y 259.043,Z 488.84,A -85,B 0,C 180,E1 -18530.632,E2 -18530.632} C_VEL
LIN {X 0,Y 257.771,Z 489.105,A -85,B 0,C 180,E1 -18532.165,E2 -18532.165} C_VEL
LIN {X 0,Y 256.776,Z 488.8,A -85,B 0,C 180,E1 -18533.715,E2 -18533.715} C_VEL
LIN {X 0,Y 255.964,Z 487.895,A -85,B 0,C 180,E1 -18535.275,E2 -18535.275} C_VEL
LIN {X 0,Y 255.181,Z 485.409,A -85,B 0,C 180,E1 -18537.632,E2 -18537.632} C_VEL
LIN {X 0,Y 254.736,Z 481.545,A -85,B 0,C 180,E1 -18540,E2 -18540} C_VEL
LIN {X 0,Y 254.668,Z 476.124,A -85,B 0,C 180,E1 -18542.373,E2 -18542.373} C_VEL
LIN {X 0,Y 254.91,Z 470.237,A -85,B 0,C 180,E1 -18544.348,E2 -18544.348} C_VEL
LIN {X 0,Y 255.323,Z 462.858,A -85,B 0,C 180,E1 -18546.321,E2 -18546.321} C_VEL
LIN {X 0,Y 255.648,Z 453.697,A -85,B 0,C 180,E1 -18548.271,E2 -18548.271} C_VEL
LIN {X 0,Y 256.07,Z 444.236,A -85,B 0,C 180,E1 -18549.877,E2 -18549.877} C_VEL
LIN {X 0,Y 256.547,Z 433.946,A -85,B 0,C 180,E1 -18551.256,E2 -18551.256} C_VEL
LIN {X 0,Y 255.321,Z 421.829,A -85,B 0,C 180,E1 -18552.519,E2 -18552.519} C_VEL
LIN {X 0,Y 254.827,Z 415.258,A -85,B 0,C 180,E1 -18553.101,E2 -18553.101} C_VEL
LIN {X 0,Y 255.086,Z 408.683,A -85,B 0,C 180,E1 -18557.642,E2 -18557.642} C_VEL
LIN {X 0,Y 255.487,Z 402.788,A -85,B 0,C 180,E1 -18561.8,E2 -18561.8} C_VEL
LIN {X 0,Y 255.943,Z 396.88,A -85,B 0,C 180,E1 -18566.063,E2 -18566.063} C_VEL
LIN {X 0,Y 256.459,Z 392.106,A -85,B 0,C 180,E1 -18569.556,E2 -18569.556} C_VEL
LIN {X 0,Y 256.41,Z 388.743,A -85,B 0,C 180,E1 -18572.101,E2 -18572.101} C_VEL
LIN {X 0,Y 256.121,Z 388.581,A -85,B 0,C 180,E1 -18577.272,E2 -18577.272} C_VEL
LIN {X 0,Y 256.058,Z 388.587,A -85,B 0,C 180,E1 -18581.203,E2 -18581.203} C_VEL
LIN {X 0,Y 256.065,Z 388.586,A -85,B 0,C 180,E1 -18585.529,E2 -18585.529} C_VEL
LIN {X 0,Y 256.058,Z 388.59,A -85,B 0,C 180,E1 -18588.797,E2 -18588.797} C_VEL
LIN {X 0,Y 256.132,Z 388.58,A -85,B 0,C 180,E1 -18592.867,E2 -18592.867} C_VEL
LIN {X 0,Y 256.07,Z 388.588,A -85,B 0,C 180,E1 -18596.707,E2 -18596.707} C_VEL
LIN {X 0,Y 256.113,Z 388.582,A -85,B 0,C 180,E1 -18600.4,E2 -18600.4} C_VEL
LIN {X 0,Y 256.191,Z 388.572,A -85,B 0,C 180,E1 -18604.861,E2 -18604.861} C_VEL
LIN {X 0,Y 256.172,Z 388.571,A -85,B 0,C 180,E1 -18609.105,E2 -18609.105} C_VEL
LIN {X 0,Y 256.303,Z 388.56,A -85,B 0,C 180,E1 -18614.085,E2 -18614.085} C_VEL
LIN {X 0,Y 256.298,Z 388.555,A -85,B 0,C 180,E1 -18617.328,E2 -18617.328} C_VEL
LIN {X 0,Y 256.519,Z 388.534,A -85,B 0,C 180,E1 -18622.126,E2 -18622.126} C_VEL
LIN {X 0,Y 256.502,Z 388.531,A -85,B 0,C 180,E1 -18626.859,E2 -18626.859} C_VEL
LIN {X 0,Y 256.768,Z 388.503,A -85,B 0,C 180,E1 -18630,E2 -18630} C_VEL
LIN {X 0,Y 256.503,Z 388.531,A -85,B 0,C 180,E1 -18633.141,E2 -18633.141} C_VEL
LIN {X 0,Y 256.541,Z 388.531,A -85,B 0,C 180,E1 -18637.873,E2 -18637.873} C_VEL
LIN {X 0,Y 256.313,Z 388.555,A -85,B 0,C 180,E1 -18641.066,E2 -18641.066} C_VEL
LIN {X 0,Y 256.303,Z 388.56,A -85,B 0,C 180,E1 -18645.915,E2 -18645.915} C_VEL
LIN {X 0,Y 256.221,Z 388.565,A -85,B 0,C 180,E1 -18650.89,E2 -18650.89} C_VEL
LIN {X 0,Y 256.191,Z 388.572,A -85,B 0,C 180,E1 -18655.138,E2 -18655.138} C_VEL
LIN {X 0,Y 256.113,Z 388.582,A -85,B 0,C 180,E1 -18659.6,E2 -18659.6} C_VEL
LIN {X 0,Y 256.087,Z 388.586,A -85,B 0,C 180,E1 -18663.29,E2 -18663.29} C_VEL
LIN {X 0,Y 256.131,Z 388.581,A -85,B 0,C 180,E1 -18667.275,E2 -18667.275} C_VEL
LIN {X 0,Y 256.059,Z 388.59,A -85,B 0,C 180,E1 -18671.203,E2 -18671.203} C_VEL
LIN {X 0,Y 256.042,Z 388.59,A -85,B 0,C 180,E1 -18675.534,E2 -18675.534} C_VEL
LIN {X 0,Y 256.056,Z 388.588,A -85,B 0,C 180,E1 -18678.796,E2 -18678.796} C_VEL
LIN {X 0,Y 256.131,Z 388.58,A -85,B 0,C 180,E1 -18682.867,E2 -18682.867} C_VEL
LIN {X 0,Y 256.069,Z 388.585,A -85,B 0,C 180,E1 -18686.707,E2 -18686.707} C_VEL
LIN {X 0,Y 256.116,Z 388.581,A -85,B 0,C 180,E1 -18690.4,E2 -18690.4} C_VEL
LIN {X 0,Y 256.19,Z 388.572,A -85,B 0,C 180,E1 -18694.861,E2 -18694.861} C_VEL
LIN {X 0,Y 256.169,Z 388.576,A -85,B 0,C 180,E1 -18699.105,E2 -18699.105} C_VEL
LIN {X 0,Y 256.302,Z 388.556,A -85,B 0,C 180,E1 -18704.085,E2 -18704.085} C_VEL
LIN {X 0,Y 256.313,Z 388.557,A -85,B 0,C 180,E1 -18708.934,E2 -18708.934} C_VEL
LIN {X 0,Y 256.542,Z 388.526,A -85,B 0,C 180,E1 -18712.127,E2 -18712.127} C_VEL
LIN {X 0,Y 256.716,Z 388.508,A -85,B 0,C 180,E1 -18718.431,E2 -18718.431} C_VEL
LIN {X 0,Y 256.719,Z 388.504,A -85,B 0,C 180,E1 -18721.569,E2 -18721.569} C_VEL
LIN {X 0,Y 256.542,Z 388.527,A -85,B 0,C 180,E1 -18727.873,E2 -18727.873} C_VEL
LIN {X 0,Y 256.311,Z 388.555,A -85,B 0,C 180,E1 -18731.066,E2 -18731.066} C_VEL
LIN {X 0,Y 256.302,Z 388.558,A -85,B 0,C 180,E1 -18735.915,E2 -18735.915} C_VEL
LIN {X 0,Y 256.168,Z 388.574,A -85,B 0,C 180,E1 -18740.895,E2 -18740.895} C_VEL
LIN {X 0,Y 256.19,Z 388.569,A -85,B 0,C 180,E1 -18745.139,E2 -18745.139} C_VEL
LIN {X 0,Y 256.105,Z 388.583,A -85,B 0,C 180,E1 -18749.601,E2 -18749.601} C_VEL
LIN {X 0,Y 256.086,Z 388.583,A -85,B 0,C 180,E1 -18753.29,E2 -18753.29} C_VEL
LIN {X 0,Y 256.129,Z 388.578,A -85,B 0,C 180,E1 -18757.275,E2 -18757.275} C_VEL
LIN {X 0,Y 256.058,Z 388.587,A -85,B 0,C 180,E1 -18761.203,E2 -18761.203} C_VEL
LIN {X 0,Y 256.061,Z 388.587,A -85,B 0,C 180,E1 -18765.365,E2 -18765.365} C_VEL
LIN {X 0,Y 255.821,Z 388.882,A -85,B 0,C 180,E1 -18766.237,E2 -18766.237} C_VEL
LIN {X 0,Y 254.743,Z 390.208,A -85,B 0,C 180,E1 -18767.505,E2 -18767.505} C_VEL
LIN {X 0,Y 253.271,Z 392.254,A -85,B 0,C 180,E1 -18768.722,E2 -18768.722} C_VEL
LIN {X 0,Y 251.469,Z 395.738,A -85,B 0,C 180,E1 -18770.343,E2 -18770.343} C_VEL
LIN {X 0,Y 250.914,Z 398.285,A -85,B 0,C 180,E1 -18771.579,E2 -18771.579} C_VEL
LIN {X 0,Y 250.984,Z 399.102,A -85,B 0,C 180,E1 -18771.997,E2 -18771.997} C_VEL
LIN {X 0,Y 252.879,Z 407.977,A -85,B 0,C 180,E1 -18776.487,E2 -18776.487} C_VEL
LIN {X 0,Y 253.677,Z 411.561,A -85,B 0,C 180,E1 -18778.238,E2 -18778.238} C_VEL
LIN {X 0,Y 253.631,Z 413.605,A -85,B 0,C 180,E1 -18779.204,E2 -18779.204} C_VEL
LIN {X 0,Y 251.047,Z 424.54,A -85,B 0,C 180,E1 -18784.284,E2 -18784.284} C_VEL
LIN {X 0,Y 248.991,Z 437.316,A -85,B 0,C 180,E1 -18790.255,E2 -18790.255} C_VEL
LIN {X 0,Y 249.15,Z 450.13,A -85,B 0,C 180,E1 -18791.071,E2 -18791.071} C_VEL
LIN {X 0,Y 249.905,Z 462.927,A -85,B 0,C 180,E1 -18792.22,E2 -18792.22} C_VEL
LIN {X 0,Y 250.581,Z 473.139,A -85,B 0,C 180,E1 -18793.406,E2 -18793.406} C_VEL
LIN {X 0,Y 249.918,Z 483.41,A -85,B 0,C 180,E1 -18794.923,E2 -18794.923} C_VEL
LIN {X 0,Y 249.217,Z 493.334,A -85,B 0,C 180,E1 -18796.754,E2 -18796.754} C_VEL
LIN {X 0,Y 248.741,Z 501.45,A -85,B 0,C 180,E1 -18798.593,E2 -18798.593} C_VEL
LIN {X 0,Y 248.375,Z 510.086,A -85,B 0,C 180,E1 -18801.047,E2 -18801.047} C_VEL
LIN {X 0,Y 248.428,Z 516.909,A -85,B 0,C 180,E1 -18803.503,E2 -18803.503} C_VEL
LIN {X 0,Y 248.498,Z 522.11,A -85,B 0,C 180,E1 -18805.946,E2 -18805.946} C_VEL
LIN {X 0,Y 248.472,Z 525.948,A -85,B 0,C 180,E1 -18808.379,E2 -18808.379} C_VEL
LIN {X 0,Y 248.342,Z 527.82,A -85,B 0,C 180,E1 -18810,E2 -18810} C_VEL
LIN {X 0,Y 248.173,Z 529.162,A -85,B 0,C 180,E1 -18811.623,E2 -18811.623} C_VEL
LIN {X 0,Y 247.834,Z 530.047,A -85,B 0,C 180,E1 -18813.251,E2 -18813.251} C_VEL
LIN {X 0,Y 247.408,Z 530.585,A -85,B 0,C 180,E1 -18816.157,E2 -18816.157} C_VEL
LIN {X 0,Y 247.376,Z 530.201,A -85,B 0,C 180,E1 -18818.167,E2 -18818.167} C_VEL
LIN {X 0,Y 247.532,Z 529.487,A -85,B 0,C 180,E1 -18819.809,E2 -18819.809} C_VEL
LIN {X 0,Y 248.45,Z 526.864,A -85,B 0,C 180,E1 -18823.079,E2 -18823.079} C_VEL
LIN {X 0,Y 249.955,Z 523.892,A -85,B 0,C 180,E1 -18825.493,E2 -18825.493} C_VEL
LIN {X 0,Y 251.782,Z 519.998,A -85,B 0,C 180,E1 -18827.881,E2 -18827.881} C_VEL
LIN {X 0,Y 254.288,Z 515.119,A -85,B 0,C 180,E1 -18830.211,E2 -18830.211} C_VEL
LIN {X 0,Y 257.959,Z 508.004,A -85,B 0,C 180,E1 -18832.845,E2 -18832.845} C_VEL
LIN {X 0,Y 261.648,Z 500.431,A -85,B 0,C 180,E1 -18835.028,E2 -18835.028} C_VEL
LIN {X 0,Y 265.889,Z 491.334,A -85,B 0,C 180,E1 -18837.127,E2 -18837.127} C_VEL
LIN {X 0,Y 268.744,Z 482.528,A -85,B 0,C 180,E1 -18838.934,E2 -18838.934} C_VEL
LIN {X 0,Y 270.535,Z 472.555,A -85,B 0,C 180,E1 -18840.988,E2 -18840.988} C_VEL
LIN {X 0,Y 271.228,Z 460.615,A -85,B 0,C 180,E1 -18843.494,E2 -18843.494} C_VEL
LIN {X 0,Y 271.057,Z 452.992,A -85,B 0,C 180,E1 -18845.203,E2 -18845.203} C_VEL
LIN {X 0,Y 270.186,Z 449.795,A -85,B 0,C 180,E1 -18846.258,E2 -18846.258} C_VEL
LIN {X 0,Y 267.31,Z 443.665,A -85,B 0,C 180,E1 -18849.124,E2 -18849.124} C_VEL
LIN {X 0,Y 264.588,Z 438.535,A -85,B 0,C 180,E1 -18852.779,E2 -18852.779} C_VEL
LIN {X 0,Y 264.053,Z 436.946,A -85,B 0,C 180,E1 -18854.059,E2 -18854.059} C_VEL
LIN {X 0,Y 263.329,Z 435.675,A -85,B 0,C 180,E1 -18856.105,E2 -18856.105} C_VEL
LIN {X 0,Y 263.073,Z 434.989,A -85,B 0,C 180,E1 -18858.42,E2 -18858.42} C_VEL
LIN {X 0,Y 263.268,Z 435.329,A -85,B 0,C 180,E1 -18860.73,E2 -18860.73} C_VEL
LIN {X 0,Y 265.034,Z 438.506,A -85,B 0,C 180,E1 -18865.29,E2 -18865.29} C_VEL
LIN {X 0,Y 266.761,Z 443.896,A -85,B 0,C 180,E1 -18868.714,E2 -18868.714} C_VEL
LIN {X 0,Y 267.818,Z 448.87,A -85,B 0,C 180,E1 -18871.037,E2 -18871.037} C_VEL
LIN {X 0,Y 268.823,Z 456.522,A -85,B 0,C 180,E1 -18874.098,E2 -18874.098} C_VEL
LIN {X 0,Y 268.948,Z 462.965,A -85,B 0,C 180,E1 -18876.475,E2 -18876.475} C_VEL
LIN {X 0,Y 268.405,Z 468.57,A -85,B 0,C 180,E1 -18878.495,E2 -18878.495} C_VEL
LIN {X 0,Y 267.699,Z 470.799,A -85,B 0,C 180,E1 -18879.242,E2 -18879.242} C_VEL
LIN {X 0,Y 263.827,Z 477.532,A -85,B 0,C 180,E1 -18881.357,E2 -18881.357} C_VEL
LIN {X 0,Y 260.283,Z 482.636,A -85,B 0,C 180,E1 -18883.53,E2 -18883.53} C_VEL
LIN {X 0,Y 257.186,Z 486.368,A -85,B 0,C 180,E1 -18885.763,E2 -18885.763} C_VEL
LIN {X 0,Y 255.387,Z 488.094,A -85,B 0,C 180,E1 -18887.282,E2 -18887.282} C_VEL
LIN {X 0,Y 253.69,Z 489.262,A -85,B 0,C 180,E1 -18888.818,E2 -18888.818} C_VEL
LIN {X 0,Y 252.115,Z 489.902,A -85,B 0,C 180,E1 -18890.372,E2 -18890.372} C_VEL
LIN {X 0,Y 250.792,Z 489.977,A -85,B 0,C 180,E1 -18891.946,E2 -18891.946} C_VEL
LIN {X 0,Y 249.761,Z 489.442,A -85,B 0,C 180,E1 -18893.537,E2 -18893.537} C_VEL
LIN {X 0,Y 248.924,Z 488.338,A -85,B 0,C 180,E1 -18895.141,E2 -18895.141} C_VEL
LIN {X 0,Y 248.102,Z 485.591,A -85,B 0,C 180,E1 -18897.565,E2 -18897.565} C_VEL
LIN {X 0,Y 247.637,Z 481.411,A -85,B 0,C 180,E1 -18900,E2 -18900} C_VEL
LIN {X 0,Y 247.584,Z 475.681,A -85,B 0,C 180,E1 -18902.441,E2 -18902.441} C_VEL
LIN {X 0,Y 247.853,Z 469.527,A -85,B 0,C 180,E1 -18904.472,E2 -18904.472} C_VEL
LIN {X 0,Y 248.259,Z 461.78,A -85,B 0,C 180,E1 -18906.502,E2 -18906.502} C_VEL
LIN {X 0,Y 248.602,Z 452.415,A -85,B 0,C 180,E1 -18908.458,E2 -18908.458} C_VEL
LIN {X 0,Y 249.102,Z 442.182,A -85,B 0,C 180,E1 -18910.156,E2 -18910.156} C_VEL
LIN {X 0,Y 249.366,Z 432.979,A -85,B 0,C 180,E1 -18911.378,E2 -18911.378} C_VEL
LIN {X 0,Y 248.061,Z 420.355,A -85,B 0,C 180,E1 -18912.684,E2 -18912.684} C_VEL
LIN {X 0,Y 247.738,Z 415.59,A -85,B 0,C 180,E1 -18913.118,E2 -18913.118} C_VEL
LIN {X 0,Y 247.998,Z 409.639,A -85,B 0,C 180,E1 -18917.311,E2 -18917.311} C_VEL
LIN {X 0,Y 248.39,Z 403.707,A -85,B 0,C 180,E1 -18921.582,E2 -18921.582} C_VEL
LIN {X 0,Y 248.861,Z 397.703,A -85,B 0,C 180,E1 -18925.999,E2 -18925.999} C_VEL
LIN {X 0,Y 249.317,Z 393.569,A -85,B 0,C 180,E1 -18929.089,E2 -18929.089} C_VEL
LIN {X 0,Y 249.537,Z 390.604,A -85,B 0,C 180,E1 -18931.334,E2 -18931.334} C_VEL
LIN {X 0,Y 249.281,Z 389.425,A -85,B 0,C 180,E1 -18932.39,E2 -18932.39} C_VEL
LIN {X 0,Y 249.074,Z 389.457,A -85,B 0,C 180,E1 -18936.338,E2 -18936.338} C_VEL
LIN {X 0,Y 249.008,Z 389.467,A -85,B 0,C 180,E1 -18940.478,E2 -18940.478} C_VEL
LIN {X 0,Y 249.01,Z 389.468,A -85,B 0,C 180,E1 -18944.878,E2 -18944.878} C_VEL
LIN {X 0,Y 249.021,Z 389.464,A -85,B 0,C 180,E1 -18947.363,E2 -18947.363} C_VEL
LIN {X 0,Y 249.046,Z 389.459,A -85,B 0,C 180,E1 -18952.2,E2 -18952.2} C_VEL
LIN {X 0,Y 249.046,Z 389.461,A -85,B 0,C 180,E1 -18955.64,E2 -18955.64} C_VEL
LIN {X 0,Y 249.053,Z 389.457,A -85,B 0,C 180,E1 -18959.473,E2 -18959.473} C_VEL
LIN {X 0,Y 249.075,Z 389.457,A -85,B 0,C 180,E1 -18963.162,E2 -18963.162} C_VEL
LIN {X 0,Y 249.084,Z 389.456,A -85,B 0,C 180,E1 -18966.733,E2 -18966.733} C_VEL
LIN {X 0,Y 249.115,Z 389.454,A -85,B 0,C 180,E1 -18970.212,E2 -18970.212} C_VEL
LIN {X 0,Y 249.245,Z 389.436,A -85,B 0,C 180,E1 -18973.622,E2 -18973.622} C_VEL
LIN {X 0,Y 249.248,Z 389.436,A -85,B 0,C 180,E1 -18978.616,E2 -18978.616} C_VEL
LIN {X 0,Y 249.458,Z 389.412,A -85,B 0,C 180,E1 -18981.902,E2 -18981.902} C_VEL
LIN {X 0,Y 249.299,Z 389.427,A -85,B 0,C 180,E1 -18985.148,E2 -18985.148} C_VEL
LIN {X 0,Y 249.679,Z 389.383,A -85,B 0,C 180,E1 -18988.387,E2 -18988.387} C_VEL
LIN {X 0,Y 249.68,Z 389.383,A -85,B 0,C 180,E1 -18991.613,E2 -18991.613} C_VEL
LIN {X 0,Y 249.463,Z 389.409,A -85,B 0,C 180,E1 -18996.47,E2 -18996.47} C_VEL
LIN {X 0,Y 249.392,Z 389.421,A -85,B 0,C 180,E1 -18999.734,E2 -18999.734} C_VEL
LIN {X 0,Y 249.209,Z 389.439,A -85,B 0,C 180,E1 -19004.703,E2 -19004.703} C_VEL
LIN {X 0,Y 249.144,Z 389.45,A -85,B 0,C 180,E1 -19008.077,E2 -19008.077} C_VEL
LIN {X 0,Y 249.107,Z 389.454,A -85,B 0,C 180,E1 -19011.516,E2 -19011.516} C_VEL
LIN {X 0,Y 249.133,Z 389.453,A -85,B 0,C 180,E1 -19015.482,E2 -19015.482} C_VEL
LIN {X 0,Y 249.082,Z 389.456,A -85,B 0,C 180,E1 -19018.992,E2 -19018.992} C_VEL
LIN {X 0,Y 249.038,Z 389.461,A -85,B 0,C 180,E1 -19022.425,E2 -19022.425} C_VEL
LIN {X 0,Y 249.071,Z 389.457,A -85,B 0,C 180,E1 -19026.338,E2 -19026.338} C_VEL
LIN {X 0,Y 249.028,Z 389.462,A -85,B 0,C 180,E1 -19030.474,E2 -19030.474} C_VEL
LIN {X 0,Y 248.987,Z 389.469,A -85,B 0,C 180,E1 -19034.883,E2 -19034.883} C_VEL
LIN {X 0,Y 249.011,Z 389.467,A -85,B 0,C 180,E1 -19037.361,E2 -19037.361} C_VEL
LIN {X 0,Y 249.027,Z 389.464,A -85,B 0,C 180,E1 -19041.619,E2 -19041.619} C_VEL
LIN {X 0,Y 249.045,Z 389.459,A -85,B 0,C 180,E1 -19045.639,E2 -19045.639} C_VEL
LIN {X 0,Y 249.054,Z 389.461,A -85,B 0,C 180,E1 -19049.473,E2 -19049.473} C_VEL
LIN {X 0,Y 249.076,Z 389.457,A -85,B 0,C 180,E1 -19053.162,E2 -19053.162} C_VEL
LIN {X 0,Y 249.082,Z 389.458,A -85,B 0,C 180,E1 -19056.733,E2 -19056.733} C_VEL
LIN {X 0,Y 249.113,Z 389.453,A -85,B 0,C 180,E1 -19060.211,E2 -19060.211} C_VEL
LIN {X 0,Y 249.244,Z 389.434,A -85,B 0,C 180,E1 -19063.622,E2 -19063.622} C_VEL
LIN {X 0,Y 249.256,Z 389.438,A -85,B 0,C 180,E1 -19068.617,E2 -19068.617} C_VEL
LIN {X 0,Y 249.486,Z 389.403,A -85,B 0,C 180,E1 -19071.903,E2 -19071.903} C_VEL
LIN {X 0,Y 249.438,Z 389.414,A -85,B 0,C 180,E1 -19076.769,E2 -19076.769} C_VEL
LIN {X 0,Y 249.731,Z 389.374,A -85,B 0,C 180,E1 -19080,E2 -19080} C_VEL
LIN {X 0,Y 249.443,Z 389.411,A -85,B 0,C 180,E1 -19083.23,E2 -19083.23} C_VEL
LIN {X 0,Y 249.486,Z 389.407,A -85,B 0,C 180,E1 -19088.097,E2 -19088.097} C_VEL
LIN {X 0,Y 249.255,Z 389.434,A -85,B 0,C 180,E1 -19091.383,E2 -19091.383} C_VEL
LIN {X 0,Y 249.243,Z 389.437,A -85,B 0,C 180,E1 -19096.378,E2 -19096.378} C_VEL
LIN {X 0,Y 249.088,Z 389.456,A -85,B 0,C 180,E1 -19101.518,E2 -19101.518} C_VEL
LIN {X 0,Y 249.132,Z 389.449,A -85,B 0,C 180,E1 -19105.482,E2 -19105.482} C_VEL
LIN {X 0,Y 249.074,Z 389.457,A -85,B 0,C 180,E1 -19108.989,E2 -19108.989} C_VEL
LIN {X 0,Y 249.037,Z 389.462,A -85,B 0,C 180,E1 -19112.425,E2 -19112.425} C_VEL
LIN {X 0,Y 249.07,Z 389.458,A -85,B 0,C 180,E1 -19116.339,E2 -19116.339} C_VEL
LIN {X 0,Y 249.027,Z 389.463,A -85,B 0,C 180,E1 -19120.474,E2 -19120.474} C_VEL
LIN {X 0,Y 249.011,Z 389.463,A -85,B 0,C 180,E1 -19124.878,E2 -19124.878} C_VEL
LIN {X 0,Y 249.092,Z 389.507,A -85,B 0,C 180,E1 -19126.905,E2 -19126.905} C_VEL
LIN {X 0,Y 250.984,Z 399.102,A -85,B 0,C 180,E1 -19131.997,E2 -19131.997} C_VEL
LIN {X 0,Y 250.828,Z 401.574,A -85,B 0,C 180,E1 -19133.22,E2 -19133.22} C_VEL
LIN {X 0,Y 248.947,Z 405.865,A -85,B 0,C 180,E1 -19135.219,E2 -19135.219} C_VEL
LIN {X 0,Y 246.707,Z 411.077,A -85,B 0,C 180,E1 -19137.661,E2 -19137.661} C_VEL
LIN {X 0,Y 246.59,Z 412.787,A -85,B 0,C 180,E1 -19138.496,E2 -19138.496} C_VEL
LIN {X 0,Y 246.053,Z 415.924,A -85,B 0,C 180,E1 -19140.01,E2 -19140.01} C_VEL
LIN {X 0,Y 243.505,Z 426.835,A -85,B 0,C 180,E1 -19145.26,E2 -19145.26} C_VEL
LIN {X 0,Y 241.899,Z 436.997,A -85,B 0,C 180,E1 -19150.205,E2 -19150.205} C_VEL
LIN {X 0,Y 242.074,Z 450.9,A -85,B 0,C 180,E1 -19151.156,E2 -19151.156} C_VEL
LIN {X 0,Y 242.927,Z 464.22,A -85,B 0,C 180,E1 -19152.433,E2 -19152.433} C_VEL
LIN {X 0,Y 243.505,Z 472.449,A -85,B 0,C 180,E1 -19153.441,E2 -19153.441} C_VEL
LIN {X 0,Y 242.827,Z 483.359,A -85,B 0,C 180,E1 -19155.116,E2 -19155.116} C_VEL
LIN {X 0,Y 242.165,Z 493.151,A -85,B 0,C 180,E1 -19157.002,E2 -19157.002} C_VEL
LIN {X 0,Y 241.684,Z 501.916,A -85,B 0,C 180,E1 -19159.105,E2 -19159.105} C_VEL
LIN {X 0,Y 241.408,Z 510.33,A -85,B 0,C 180,E1 -19161.63,E2 -19161.63} C_VEL
LIN {X 0,Y 241.473,Z 516.862,A -85,B 0,C 180,E1 -19164.153,E2 -19164.153} C_VEL
LIN {X 0,Y 241.543,Z 521.861,A -85,B 0,C 180,E1 -19166.664,E2 -19166.664} C_VEL
LIN {X 0,Y 241.516,Z 524.428,A -85,B 0,C 180,E1 -19168.333,E2 -19168.333} C_VEL
LIN {X 0,Y 241.383,Z 526.418,A -85,B 0,C 180,E1 -19170,E2 -19170} C_VEL
LIN {X 0,Y 241.171,Z 527.918,A -85,B 0,C 180,E1 -19171.67,E2 -19171.67} C_VEL
LIN {X 0,Y 240.8,Z 528.898,A -85,B 0,C 180,E1 -19173.347,E2 -19173.347} C_VEL
LIN {X 0,Y 240.362,Z 529.659,A -85,B 0,C 180,E1 -19176.717,E2 -19176.717} C_VEL
LIN {X 0,Y 240.511,Z 528.829,A -85,B 0,C 180,E1 -19180.098,E2 -19180.098} C_VEL
LIN {X 0,Y 241.515,Z 526.529,A -85,B 0,C 180,E1 -19183.462,E2 -19183.462} C_VEL
LIN {X 0,Y 243.632,Z 522.672,A -85,B 0,C 180,E1 -19186.766,E2 -19186.766} C_VEL
LIN {X 0,Y 246.514,Z 517.583,A -85,B 0,C 180,E1 -19189.811,E2 -19189.811} C_VEL
LIN {X 0,Y 249.734,Z 511.909,A -85,B 0,C 180,E1 -19192.329,E2 -19192.329} C_VEL
LIN {X 0,Y 253.928,Z 504.322,A -85,B 0,C 180,E1 -19194.966,E2 -19194.966} C_VEL
LIN {X 0,Y 258.257,Z 496.217,A -85,B 0,C 180,E1 -19197.118,E2 -19197.118} C_VEL
LIN {X 0,Y 261.752,Z 488.358,A -85,B 0,C 180,E1 -19198.901,E2 -19198.901} C_VEL
LIN {X 0,Y 263.85,Z 481.52,A -85,B 0,C 180,E1 -19200.404,E2 -19200.404} C_VEL
LIN {X 0,Y 265.686,Z 471.345,A -85,B 0,C 180,E1 -19202.667,E2 -19202.667} C_VEL
LIN {X 0,Y 266.454,Z 462.439,A -85,B 0,C 180,E1 -19204.692,E2 -19204.692} C_VEL
LIN {X 0,Y 266.641,Z 457.574,A -85,B 0,C 180,E1 -19205.875,E2 -19205.875} C_VEL
LIN {X 0,Y 265.855,Z 454.838,A -85,B 0,C 180,E1 -19206.883,E2 -19206.883} C_VEL
LIN {X 0,Y 263.473,Z 449.105,A -85,B 0,C 180,E1 -19209.806,E2 -19209.806} C_VEL
LIN {X 0,Y 261.299,Z 444.308,A -85,B 0,C 180,E1 -19213.431,E2 -19213.431} C_VEL
LIN {X 0,Y 260.974,Z 443.203,A -85,B 0,C 180,E1 -19214.442,E2 -19214.442} C_VEL
LIN {X 0,Y 260.208,Z 441.681,A -85,B 0,C 180,E1 -19217.528,E2 -19217.528} C_VEL
LIN {X 0,Y 260.18,Z 441.468,A -85,B 0,C 180,E1 -19219.587,E2 -19219.587} C_VEL
LIN {X 0,Y 260.311,Z 442.281,A -85,B 0,C 180,E1 -19221.613,E2 -19221.613} C_VEL
LIN {X 0,Y 260.928,Z 443.729,A -85,B 0,C 180,E1 -19223.905,E2 -19223.905} C_VEL
LIN {X 0,Y 261.629,Z 445.379,A -85,B 0,C 180,E1 -19225.659,E2 -19225.659} C_VEL
LIN {X 0,Y 262.543,Z 449.031,A -85,B 0,C 180,E1 -19228.153,E2 -19228.153} C_VEL
LIN {X 0,Y 263.178,Z 453.592,A -85,B 0,C 180,E1 -19230.477,E2 -19230.477} C_VEL
LIN {X 0,Y 263.575,Z 459.407,A -85,B 0,C 180,E1 -19233.045,E2 -19233.045} C_VEL
LIN {X 0,Y 263.443,Z 465.721,A -85,B 0,C 180,E1 -19235.609,E2 -19235.609} C_VEL
LIN {X 0,Y 262.505,Z 471.722,A -85,B 0,C 180,E1 -19237.987,E2 -19237.987} C_VEL
LIN {X 0,Y 261.512,Z 473.909,A -85,B 0,C 180,E1 -19238.727,E2 -19238.727} C_VEL
LIN {X 0,Y 257.414,Z 480.038,A -85,B 0,C 180,E1 -19240.875,E2 -19240.875} C_VEL
LIN {X 0,Y 253.729,Z 484.75,A -85,B 0,C 180,E1 -19243.092,E2 -19243.092} C_VEL
LIN {X 0,Y 250.491,Z 488.032,A -85,B 0,C 180,E1 -19245.374,E2 -19245.374} C_VEL
LIN {X 0,Y 248.611,Z 489.524,A -85,B 0,C 180,E1 -19246.929,E2 -19246.929} C_VEL
LIN {X 0,Y 246.826,Z 490.501,A -85,B 0,C 180,E1 -19248.503,E2 -19248.503} C_VEL
LIN {X 0,Y 245.185,Z 490.913,A -85,B 0,C 180,E1 -19250.097,E2 -19250.097} C_VEL
LIN {X 0,Y 243.817,Z 490.745,A -85,B 0,C 180,E1 -19251.714,E2 -19251.714} C_VEL
LIN {X 0,Y 242.737,Z 490.023,A -85,B 0,C 180,E1 -19253.35,E2 -19253.35} C_VEL
LIN {X 0,Y 241.887,Z 488.722,A -85,B 0,C 180,E1 -19255,E2 -19255} C_VEL
LIN {X 0,Y 241.008,Z 485.651,A -85,B 0,C 180,E1 -19257.493,E2 -19257.493} C_VEL
LIN {X 0,Y 240.541,Z 481.182,A -85,B 0,C 180,E1 -19260,E2 -19260} C_VEL
LIN {X 0,Y 240.504,Z 475.099,A -85,B 0,C 180,E1 -19262.512,E2 -19262.512} C_VEL
LIN {X 0,Y 240.8,Z 468.637,A -85,B 0,C 180,E1 -19264.604,E2 -19264.604} C_VEL
LIN {X 0,Y 241.162,Z 462.348,A -85,B 0,C 180,E1 -19266.274,E2 -19266.274} C_VEL
LIN {X 0,Y 241.436,Z 453.737,A -85,B 0,C 180,E1 -19268.147,E2 -19268.147} C_VEL
LIN {X 0,Y 241.912,Z 444.107,A -85,B 0,C 180,E1 -19269.828,E2 -19269.828} C_VEL
LIN {X 0,Y 242.308,Z 433.609,A -85,B 0,C 180,E1 -19271.29,E2 -19271.29} C_VEL
LIN {X 0,Y 240.999,Z 421.067,A -85,B 0,C 180,E1 -19272.634,E2 -19272.634} C_VEL
LIN {X 0,Y 240.668,Z 415.973,A -85,B 0,C 180,E1 -19273.08,E2 -19273.08} C_VEL
LIN {X 0,Y 240.945,Z 409.389,A -85,B 0,C 180,E1 -19277.835,E2 -19277.835} C_VEL
LIN {X 0,Y 241.373,Z 403.413,A -85,B 0,C 180,E1 -19282.242,E2 -19282.242} C_VEL
LIN {X 0,Y 241.917,Z 397.413,A -85,B 0,C 180,E1 -19286.763,E2 -19286.763} C_VEL
LIN {X 0,Y 242.425,Z 392.571,A -85,B 0,C 180,E1 -19290.487,E2 -19290.487} C_VEL
LIN {X 0,Y 242.251,Z 390.3,A -85,B 0,C 180,E1 -19292.389,E2 -19292.389} C_VEL
LIN {X 0,Y 242.06,Z 390.33,A -85,B 0,C 180,E1 -19295.614,E2 -19295.614} C_VEL
LIN {X 0,Y 241.959,Z 390.343,A -85,B 0,C 180,E1 -19299.719,E2 -19299.719} C_VEL
LIN {X 0,Y 241.937,Z 390.345,A -85,B 0,C 180,E1 -19304.201,E2 -19304.201} C_VEL
LIN {X 0,Y 241.941,Z 390.346,A -85,B 0,C 180,E1 -19308.078,E2 -19308.078} C_VEL
LIN {X 0,Y 241.989,Z 390.34,A -85,B 0,C 180,E1 -19312.418,E2 -19312.418} C_VEL
LIN {X 0,Y 241.983,Z 390.344,A -85,B 0,C 180,E1 -19316.507,E2 -19316.507} C_VEL
LIN {X 0,Y 242.038,Z 390.335,A -85,B 0,C 180,E1 -19320.588,E2 -19320.588} C_VEL
LIN {X 0,Y 242.07,Z 390.332,A -85,B 0,C 180,E1 -19324.183,E2 -19324.183} C_VEL
LIN {X 0,Y 242.057,Z 390.333,A -85,B 0,C 180,E1 -19328.297,E2 -19328.297} C_VEL
LIN {X 0,Y 242.166,Z 390.318,A -85,B 0,C 180,E1 -19333.278,E2 -19333.278} C_VEL
LIN {X 0,Y 242.184,Z 390.318,A -85,B 0,C 180,E1 -19338.28,E2 -19338.28} C_VEL
LIN {X 0,Y 242.404,Z 390.289,A -85,B 0,C 180,E1 -19341.665,E2 -19341.665} C_VEL
LIN {X 0,Y 242.26,Z 390.304,A -85,B 0,C 180,E1 -19345.007,E2 -19345.007} C_VEL
LIN {X 0,Y 242.639,Z 390.261,A -85,B 0,C 180,E1 -19348.34,E2 -19348.34} C_VEL
LIN {X 0,Y 242.64,Z 390.26,A -85,B 0,C 180,E1 -19351.66,E2 -19351.66} C_VEL
LIN {X 0,Y 242.435,Z 390.284,A -85,B 0,C 180,E1 -19356.659,E2 -19356.659} C_VEL
LIN {X 0,Y 242.317,Z 390.301,A -85,B 0,C 180,E1 -19360.022,E2 -19360.022} C_VEL
LIN {X 0,Y 242.17,Z 390.317,A -85,B 0,C 180,E1 -19365.141,E2 -19365.141} C_VEL
LIN {X 0,Y 242.083,Z 390.328,A -85,B 0,C 180,E1 -19368.623,E2 -19368.623} C_VEL
LIN {X 0,Y 242.053,Z 390.331,A -85,B 0,C 180,E1 -19372.176,E2 -19372.176} C_VEL
LIN {X 0,Y 242.069,Z 390.332,A -85,B 0,C 180,E1 -19375.838,E2 -19375.838} C_VEL
LIN {X 0,Y 242.031,Z 390.335,A -85,B 0,C 180,E1 -19379.58,E2 -19379.58} C_VEL
LIN {X 0,Y 241.993,Z 390.343,A -85,B 0,C 180,E1 -19383.491,E2 -19383.491} C_VEL
LIN {X 0,Y 242.005,Z 390.338,A -85,B 0,C 180,E1 -19387.579,E2 -19387.579} C_VEL
LIN {X 0,Y 241.94,Z 390.346,A -85,B 0,C 180,E1 -19391.922,E2 -19391.922} C_VEL
LIN {X 0,Y 241.927,Z 390.346,A -85,B 0,C 180,E1 -19396.573,E2 -19396.573} C_VEL
LIN {X 0,Y 241.958,Z 390.343,A -85,B 0,C 180,E1 -19400.281,E2 -19400.281} C_VEL
LIN {X 0,Y 241.982,Z 390.34,A -85,B 0,C 180,E1 -19404.488,E2 -19404.488} C_VEL
LIN {X 0,Y 241.977,Z 390.341,A -85,B 0,C 180,E1 -19408.48,E2 -19408.48} C_VEL
LIN {X 0,Y 242.011,Z 390.337,A -85,B 0,C 180,E1 -19412.313,E2 -19412.313} C_VEL
LIN {X 0,Y 242.059,Z 390.33,A -85,B 0,C 180,E1 -19416.016,E2 -19416.016} C_VEL
LIN {X 0,Y 242.04,Z 390.333,A -85,B 0,C 180,E1 -19419.608,E2 -19419.608} C_VEL
LIN {X 0,Y 242.165,Z 390.317,A -85,B 0,C 180,E1 -19423.278,E2 -19423.278} C_VEL
LIN {X 0,Y 242.189,Z 390.316,A -85,B 0,C 180,E1 -19428.28,E2 -19428.28} C_VEL
LIN {X 0,Y 242.437,Z 390.281,A -85,B 0,C 180,E1 -19431.666,E2 -19431.666} C_VEL
LIN {X 0,Y 242.262,Z 390.307,A -85,B 0,C 180,E1 -19435.007,E2 -19435.007} C_VEL
LIN {X 0,Y 242.638,Z 390.261,A -85,B 0,C 180,E1 -19438.34,E2 -19438.34} C_VEL
LIN {X 0,Y 242.641,Z 390.257,A -85,B 0,C 180,E1 -19441.66,E2 -19441.66} C_VEL
LIN {X 0,Y 242.436,Z 390.285,A -85,B 0,C 180,E1 -19446.659,E2 -19446.659} C_VEL
LIN {X 0,Y 242.347,Z 390.295,A -85,B 0,C 180,E1 -19450.02,E2 -19450.02} C_VEL
LIN {X 0,Y 242.169,Z 390.316,A -85,B 0,C 180,E1 -19455.141,E2 -19455.141} C_VEL
LIN {X 0,Y 242.075,Z 390.33,A -85,B 0,C 180,E1 -19458.624,E2 -19458.624} C_VEL
LIN {X 0,Y 242.014,Z 390.34,A -85,B 0,C 180,E1 -19462.18,E2 -19462.18} C_VEL
LIN {X 0,Y 242.068,Z 390.33,A -85,B 0,C 180,E1 -19465.838,E2 -19465.838} C_VEL
LIN {X 0,Y 242.008,Z 390.339,A -85,B 0,C 180,E1 -19469.583,E2 -19469.583} C_VEL
LIN {X 0,Y 241.992,Z 390.339,A -85,B 0,C 180,E1 -19473.491,E2 -19473.491} C_VEL
LIN {X 0,Y 242.003,Z 390.34,A -85,B 0,C 180,E1 -19477.579,E2 -19477.579} C_VEL
LIN {X 0,Y 241.945,Z 390.346,A -85,B 0,C 180,E1 -19481.921,E2 -19481.921} C_VEL
LIN {X 0,Y 242.086,Z 390.518,A -85,B 0,C 180,E1 -19486.685,E2 -19486.685} C_VEL
LIN {X 0,Y 243.628,Z 398.645,A -85,B 0,C 180,E1 -19491.158,E2 -19491.158} C_VEL
LIN {X 0,Y 245.622,Z 407.997,A -85,B 0,C 180,E1 -19496.076,E2 -19496.076} C_VEL
LIN {X 0,Y 246.59,Z 412.787,A -85,B 0,C 180,E1 -19498.496,E2 -19498.496} C_VEL
LIN {X 0,Y 246.281,Z 414.477,A -85,B 0,C 180,E1 -19499.311,E2 -19499.311} C_VEL
LIN {X 0,Y 244.581,Z 417.013,A -85,B 0,C 180,E1 -19500.49,E2 -19500.49} C_VEL
LIN {X 0,Y 237.879,Z 423.617,A -85,B 0,C 180,E1 -19503.594,E2 -19503.594} C_VEL
LIN {X 0,Y 236.539,Z 426.19,A -85,B 0,C 180,E1 -19504.87,E2 -19504.87} C_VEL
LIN {X 0,Y 234.811,Z 436.745,A -85,B 0,C 180,E1 -19510.209,E2 -19510.209} C_VEL
LIN {X 0,Y 234.911,Z 448.826,A -85,B 0,C 180,E1 -19511.034,E2 -19511.034} C_VEL
LIN {X 0,Y 235.617,Z 460.804,A -85,B 0,C 180,E1 -19512.161,E2 -19512.161} C_VEL
LIN {X 0,Y 236.416,Z 472.486,A -85,B 0,C 180,E1 -19513.596,E2 -19513.596} C_VEL
LIN {X 0,Y 235.748,Z 483.191,A -85,B 0,C 180,E1 -19515.321,E2 -19515.321} C_VEL
LIN {X 0,Y 235.172,Z 491.863,A -85,B 0,C 180,E1 -19517.048,E2 -19517.048} C_VEL
LIN {X 0,Y 234.704,Z 500.733,A -85,B 0,C 180,E1 -19519.214,E2 -19519.214} C_VEL
LIN {X 0,Y 234.437,Z 508.564,A -85,B 0,C 180,E1 -19521.604,E2 -19521.604} C_VEL
LIN {X 0,Y 234.519,Z 514.839,A -85,B 0,C 180,E1 -19523.979,E2 -19523.979} C_VEL
LIN {X 0,Y 234.599,Z 520.093,A -85,B 0,C 180,E1 -19526.565,E2 -19526.565} C_VEL
LIN {X 0,Y 234.472,Z 523.936,A -85,B 0,C 180,E1 -19529.141,E2 -19529.141} C_VEL
LIN {X 0,Y 234.207,Z 526.566,A -85,B 0,C 180,E1 -19531.72,E2 -19531.72} C_VEL
LIN {X 0,Y 233.778,Z 527.686,A -85,B 0,C 180,E1 -19533.447,E2 -19533.447} C_VEL
LIN {X 0,Y 233.361,Z 528.649,A -85,B 0,C 180,E1 -19536.36,E2 -19536.36} C_VEL
LIN {X 0,Y 233.296,Z 528.599,A -85,B 0,C 180,E1 -19538.663,E2 -19538.663} C_VEL
LIN {X 0,Y 233.89,Z 527.317,A -85,B 0,C 180,E1 -19542.142,E2 -19542.142} C_VEL
LIN {X 0,Y 235.651,Z 524.565,A -85,B 0,C 180,E1 -19545.57,E2 -19545.57} C_VEL
LIN {X 0,Y 237.535,Z 521.501,A -85,B 0,C 180,E1 -19548.1,E2 -19548.1} C_VEL
LIN {X 0,Y 240.074,Z 517.517,A -85,B 0,C 180,E1 -19550.567,E2 -19550.567} C_VEL
LIN {X 0,Y 243.213,Z 512.598,A -85,B 0,C 180,E1 -19552.961,E2 -19552.961} C_VEL
LIN {X 0,Y 247.582,Z 505.407,A -85,B 0,C 180,E1 -19555.652,E2 -19555.652} C_VEL
LIN {X 0,Y 252.083,Z 497.865,A -85,B 0,C 180,E1 -19557.839,E2 -19557.839} C_VEL
LIN {X 0,Y 255.814,Z 490.511,A -85,B 0,C 180,E1 -19559.638,E2 -19559.638} C_VEL
LIN {X 0,Y 258.15,Z 484.047,A -85,B 0,C 180,E1 -19561.149,E2 -19561.149} C_VEL
LIN {X 0,Y 260.182,Z 475.766,A -85,B 0,C 180,E1 -19563.137,E2 -19563.137} C_VEL
LIN {X 0,Y 261.546,Z 467.148,A -85,B 0,C 180,E1 -19565.239,E2 -19565.239} C_VEL
LIN {X 0,Y 262.004,Z 461.853,A -85,B 0,C 180,E1 -19566.612,E2 -19566.612} C_VEL
LIN {X 0,Y 260.865,Z 458.262,A -85,B 0,C 180,E1 -19568.291,E2 -19568.291} C_VEL
LIN {X 0,Y 260.017,Z 455.57,A -85,B 0,C 180,E1 -19569.698,E2 -19569.698} C_VEL
LIN {X 0,Y 257.846,Z 450.326,A -85,B 0,C 180,E1 -19573.767,E2 -19573.767} C_VEL
LIN {X 0,Y 257.475,Z 449.053,A -85,B 0,C 180,E1 -19575.21,E2 -19575.21} C_VEL
LIN {X 0,Y 256.977,Z 447.967,A -85,B 0,C 180,E1 -19577.597,E2 -19577.597} C_VEL
LIN {X 0,Y 256.833,Z 447.902,A -85,B 0,C 180,E1 -19580.014,E2 -19580.014} C_VEL
LIN {X 0,Y 257.083,Z 449.331,A -85,B 0,C 180,E1 -19583.028,E2 -19583.028} C_VEL
LIN {X 0,Y 257.796,Z 451.694,A -85,B 0,C 180,E1 -19585.785,E2 -19585.785} C_VEL
LIN {X 0,Y 258.314,Z 455.184,A -85,B 0,C 180,E1 -19588.255,E2 -19588.255} C_VEL
LIN {X 0,Y 258.459,Z 459.821,A -85,B 0,C 180,E1 -19590.695,E2 -19590.695} C_VEL
LIN {X 0,Y 258.303,Z 465.383,A -85,B 0,C 180,E1 -19593.325,E2 -19593.325} C_VEL
LIN {X 0,Y 257.522,Z 471.091,A -85,B 0,C 180,E1 -19595.835,E2 -19595.835} C_VEL
LIN {X 0,Y 256.557,Z 474.762,A -85,B 0,C 180,E1 -19597.449,E2 -19597.449} C_VEL
LIN {X 0,Y 253.822,Z 478.946,A -85,B 0,C 180,E1 -19598.903,E2 -19598.903} C_VEL
LIN {X 0,Y 249.71,Z 484.094,A -85,B 0,C 180,E1 -19601.115,E2 -19601.115} C_VEL
LIN {X 0,Y 246.024,Z 487.852,A -85,B 0,C 180,E1 -19603.402,E2 -19603.402} C_VEL
LIN {X 0,Y 243.819,Z 489.664,A -85,B 0,C 180,E1 -19604.964,E2 -19604.964} C_VEL
LIN {X 0,Y 241.836,Z 490.924,A -85,B 0,C 180,E1 -19606.556,E2 -19606.556} C_VEL
LIN {X 0,Y 239.967,Z 491.639,A -85,B 0,C 180,E1 -19608.17,E2 -19608.17} C_VEL
LIN {X 0,Y 238.25,Z 491.831,A -85,B 0,C 180,E1 -19609.806,E2 -19609.806} C_VEL
LIN {X 0,Y 236.846,Z 491.464,A -85,B 0,C 180,E1 -19611.468,E2 -19611.468} C_VEL
LIN {X 0,Y 235.717,Z 490.52,A -85,B 0,C 180,E1 -19613.151,E2 -19613.151} C_VEL
LIN {X 0,Y 234.462,Z 488.023,A -85,B 0,C 180,E1 -19615.702,E2 -19615.702} C_VEL
LIN {X 0,Y 233.695,Z 484.192,A -85,B 0,C 180,E1 -19618.277,E2 -19618.277} C_VEL
LIN {X 0,Y 233.401,Z 478.905,A -85,B 0,C 180,E1 -19620.863,E2 -19620.863} C_VEL
LIN {X 0,Y 233.517,Z 471.894,A -85,B 0,C 180,E1 -19623.451,E2 -19623.451} C_VEL
LIN {X 0,Y 233.977,Z 464.476,A -85,B 0,C 180,E1 -19625.602,E2 -19625.602} C_VEL
LIN {X 0,Y 234.256,Z 455.368,A -85,B 0,C 180,E1 -19627.713,E2 -19627.713} C_VEL
LIN {X 0,Y 234.705,Z 445.899,A -85,B 0,C 180,E1 -19629.48,E2 -19629.48} C_VEL
LIN {X 0,Y 235.24,Z 435.924,A -85,B 0,C 180,E1 -19630.98,E2 -19630.98} C_VEL
LIN {X 0,Y 234.307,Z 425.292,A -85,B 0,C 180,E1 -19632.23,E2 -19632.23} C_VEL
LIN {X 0,Y 233.579,Z 416.258,A -85,B 0,C 180,E1 -19633.097,E2 -19633.097} C_VEL
LIN {X 0,Y 233.849,Z 410.308,A -85,B 0,C 180,E1 -19637.49,E2 -19637.49} C_VEL
LIN {X 0,Y 234.236,Z 404.923,A -85,B 0,C 180,E1 -19641.545,E2 -19641.545} C_VEL
LIN {X 0,Y 234.735,Z 399.029,A -85,B 0,C 180,E1 -19646.076,E2 -19646.076} C_VEL
LIN {X 0,Y 235.369,Z 393.372,A -85,B 0,C 180,E1 -19650.505,E2 -19650.505} C_VEL
LIN {X 0,Y 235.204,Z 391.178,A -85,B 0,C 180,E1 -19652.411,E2 -19652.411} C_VEL
LIN {X 0,Y 234.949,Z 391.219,A -85,B 0,C 180,E1 -19656.746,E2 -19656.746} C_VEL
LIN {X 0,Y 234.944,Z 391.221,A -85,B 0,C 180,E1 -19658.944,E2 -19658.944} C_VEL
LIN {X 0,Y 234.892,Z 391.222,A -85,B 0,C 180,E1 -19663.485,E2 -19663.485} C_VEL
LIN {X 0,Y 234.892,Z 391.226,A -85,B 0,C 180,E1 -19666.515,E2 -19666.515} C_VEL
LIN {X 0,Y 234.921,Z 391.219,A -85,B 0,C 180,E1 -19671.079,E2 -19671.079} C_VEL
LIN {X 0,Y 234.93,Z 391.219,A -85,B 0,C 180,E1 -19675.362,E2 -19675.362} C_VEL
LIN {X 0,Y 234.934,Z 391.216,A -85,B 0,C 180,E1 -19679.432,E2 -19679.432} C_VEL
LIN {X 0,Y 234.997,Z 391.211,A -85,B 0,C 180,E1 -19683.794,E2 -19683.794} C_VEL
LIN {X 0,Y 235.015,Z 391.207,A -85,B 0,C 180,E1 -19688.97,E2 -19688.97} C_VEL
LIN {X 0,Y 235.099,Z 391.198,A -85,B 0,C 180,E1 -19693.059,E2 -19693.059} C_VEL
LIN {X 0,Y 235.118,Z 391.195,A -85,B 0,C 180,E1 -19697.922,E2 -19697.922} C_VEL
LIN {X 0,Y 235.334,Z 391.169,A -85,B 0,C 180,E1 -19701.412,E2 -19701.412} C_VEL
LIN {X 0,Y 235.377,Z 391.163,A -85,B 0,C 180,E1 -19703.14,E2 -19703.14} C_VEL
LIN {X 0,Y 235.599,Z 391.138,A -85,B 0,C 180,E1 -19708.29,E2 -19708.29} C_VEL
LIN {X 0,Y 235.6,Z 391.138,A -85,B 0,C 180,E1 -19711.709,E2 -19711.709} C_VEL
LIN {X 0,Y 235.406,Z 391.159,A -85,B 0,C 180,E1 -19716.858,E2 -19716.858} C_VEL
LIN {X 0,Y 235.241,Z 391.181,A -85,B 0,C 180,E1 -19720.326,E2 -19720.326} C_VEL
LIN {X 0,Y 235.117,Z 391.198,A -85,B 0,C 180,E1 -19725.606,E2 -19725.606} C_VEL
LIN {X 0,Y 235.023,Z 391.208,A -85,B 0,C 180,E1 -19729.204,E2 -19729.204} C_VEL
LIN {X 0,Y 234.984,Z 391.211,A -85,B 0,C 180,E1 -19732.88,E2 -19732.88} C_VEL
LIN {X 0,Y 234.971,Z 391.214,A -85,B 0,C 180,E1 -19736.657,E2 -19736.657} C_VEL
LIN {X 0,Y 234.934,Z 391.216,A -85,B 0,C 180,E1 -19740.567,E2 -19740.567} C_VEL
LIN {X 0,Y 234.963,Z 391.215,A -85,B 0,C 180,E1 -19744.633,E2 -19744.633} C_VEL
LIN {X 0,Y 234.943,Z 391.216,A -85,B 0,C 180,E1 -19748.944,E2 -19748.944} C_VEL
LIN {X 0,Y 234.88,Z 391.228,A -85,B 0,C 180,E1 -19753.488,E2 -19753.488} C_VEL
LIN {X 0,Y 234.88,Z 391.224,A -85,B 0,C 180,E1 -19756.512,E2 -19756.512} C_VEL
LIN {X 0,Y 234.92,Z 391.224,A -85,B 0,C 180,E1 -19761.079,E2 -19761.079} C_VEL
LIN {X 0,Y 234.928,Z 391.219,A -85,B 0,C 180,E1 -19765.361,E2 -19765.361} C_VEL
LIN {X 0,Y 234.933,Z 391.22,A -85,B 0,C 180,E1 -19769.432,E2 -19769.432} C_VEL
LIN {X 0,Y 234.996,Z 391.208,A -85,B 0,C 180,E1 -19773.793,E2 -19773.793} C_VEL
LIN {X 0,Y 235.013,Z 391.212,A -85,B 0,C 180,E1 -19778.97,E2 -19778.97} C_VEL
LIN {X 0,Y 235.098,Z 391.198,A -85,B 0,C 180,E1 -19783.059,E2 -19783.059} C_VEL
LIN {X 0,Y 235.15,Z 391.192,A -85,B 0,C 180,E1 -19787.924,E2 -19787.924} C_VEL
LIN {X 0,Y 235.392,Z 391.159,A -85,B 0,C 180,E1 -19791.414,E2 -19791.414} C_VEL
LIN {X 0,Y 235.408,Z 391.16,A -85,B 0,C 180,E1 -19793.141,E2 -19793.141} C_VEL
LIN {X 0,Y 235.598,Z 391.138,A -85,B 0,C 180,E1 -19798.29,E2 -19798.29} C_VEL
LIN {X 0,Y 235.601,Z 391.134,A -85,B 0,C 180,E1 -19801.709,E2 -19801.709} C_VEL
LIN {X 0,Y 235.408,Z 391.159,A -85,B 0,C 180,E1 -19806.858,E2 -19806.858} C_VEL
LIN {X 0,Y 235.255,Z 391.181,A -85,B 0,C 180,E1 -19810.326,E2 -19810.326} C_VEL
LIN {X 0,Y 235.116,Z 391.195,A -85,B 0,C 180,E1 -19815.606,E2 -19815.606} C_VEL
LIN {X 0,Y 235.011,Z 391.208,A -85,B 0,C 180,E1 -19819.205,E2 -19819.205} C_VEL
LIN {X 0,Y 234.963,Z 391.215,A -85,B 0,C 180,E1 -19822.883,E2 -19822.883} C_VEL
LIN {X 0,Y 234.969,Z 391.213,A -85,B 0,C 180,E1 -19826.657,E2 -19826.657} C_VEL
LIN {X 0,Y 234.924,Z 391.22,A -85,B 0,C 180,E1 -19830.569,E2 -19830.569} C_VEL
LIN {X 0,Y 234.962,Z 391.213,A -85,B 0,C 180,E1 -19834.633,E2 -19834.633} C_VEL
LIN {X 0,Y 234.942,Z 391.218,A -85,B 0,C 180,E1 -19838.944,E2 -19838.944} C_VEL
LIN {X 0,Y 234.891,Z 391.223,A -85,B 0,C 180,E1 -19843.485,E2 -19843.485} C_VEL
LIN {X 0,Y 235.017,Z 391.358,A -85,B 0,C 180,E1 -19846.397,E2 -19846.397} C_VEL
LIN {X 0,Y 236.737,Z 400.236,A -85,B 0,C 180,E1 -19851.433,E2 -19851.433} C_VEL
LIN {X 0,Y 238.78,Z 409.612,A -85,B 0,C 180,E1 -19856.505,E2 -19856.505} C_VEL
LIN {X 0,Y 239.496,Z 413.191,A -85,B 0,C 180,E1 -19858.373,E2 -19858.373} C_VEL
LIN {X 0,Y 238.896,Z 416.416,A -85,B 0,C 180,E1 -19859.992,E2 -19859.992} C_VEL
LIN {X 0,Y 236.539,Z 426.19,A -85,B 0,C 180,E1 -19864.87,E2 -19864.87} C_VEL
LIN {X 0,Y 235.513,Z 427.87,A -85,B 0,C 180,E1 -19865.709,E2 -19865.709} C_VEL
LIN {X 0,Y 232.152,Z 430.397,A -85,B 0,C 180,E1 -19867.002,E2 -19867.002} C_VEL
LIN {X 0,Y 228.855,Z 432.911,A -85,B 0,C 180,E1 -19868.331,E2 -19868.331} C_VEL
LIN {X 0,Y 227.957,Z 434.566,A -85,B 0,C 180,E1 -19869.214,E2 -19869.214} C_VEL
LIN {X 0,Y 227.719,Z 436.451,A -85,B 0,C 180,E1 -19870.213,E2 -19870.213} C_VEL
LIN {X 0,Y 227.817,Z 448.766,A -85,B 0,C 180,E1 -19871.1,E2 -19871.1} C_VEL
LIN {X 0,Y 228.59,Z 461.627,A -85,B 0,C 180,E1 -19872.382,E2 -19872.382} C_VEL
LIN {X 0,Y 229.34,Z 472.307,A -85,B 0,C 180,E1 -19873.762,E2 -19873.762} C_VEL
LIN {X 0,Y 228.673,Z 482.89,A -85,B 0,C 180,E1 -19875.54,E2 -19875.54} C_VEL
LIN {X 0,Y 228.104,Z 492.475,A -85,B 0,C 180,E1 -19877.545,E2 -19877.545} C_VEL
LIN {X 0,Y 227.665,Z 501.005,A -85,B 0,C 180,E1 -19879.776,E2 -19879.776} C_VEL
LIN {X 0,Y 227.529,Z 509.185,A -85,B 0,C 180,E1 -19882.435,E2 -19882.435} C_VEL
LIN {X 0,Y 227.57,Z 514.672,A -85,B 0,C 180,E1 -19884.684,E2 -19884.684} C_VEL
LIN {X 0,Y 227.672,Z 519.734,A -85,B 0,C 180,E1 -19887.346,E2 -19887.346} C_VEL
LIN {X 0,Y 227.511,Z 523.397,A -85,B 0,C 180,E1 -19890,E2 -19890} C_VEL
LIN {X 0,Y 227.232,Z 525.172,A -85,B 0,C 180,E1 -19891.773,E2 -19891.773} C_VEL
LIN {X 0,Y 226.774,Z 526.394,A -85,B 0,C 180,E1 -19893.554,E2 -19893.554} C_VEL
LIN {X 0,Y 226.294,Z 527.667,A -85,B 0,C 180,E1 -19897.136,E2 -19897.136} C_VEL
LIN {X 0,Y 226.497,Z 527.389,A -85,B 0,C 180,E1 -19900.73,E2 -19900.73} C_VEL
LIN {X 0,Y 227.697,Z 525.687,A -85,B 0,C 180,E1 -19904.296,E2 -19904.296} C_VEL
LIN {X 0,Y 230.033,Z 522.492,A -85,B 0,C 180,E1 -19907.79,E2 -19907.79} C_VEL
LIN {X 0,Y 232.795,Z 518.7,A -85,B 0,C 180,E1 -19910.629,E2 -19910.629} C_VEL
LIN {X 0,Y 236.729,Z 513.197,A -85,B 0,C 180,E1 -19913.628,E2 -19913.628} C_VEL
LIN {X 0,Y 242.017,Z 505.443,A -85,B 0,C 180,E1 -19916.751,E2 -19916.751} C_VEL
LIN {X 0,Y 247.598,Z 496.754,A -85,B 0,C 180,E1 -19919.317,E2 -19919.317} C_VEL
LIN {X 0,Y 251.298,Z 489.599,A -85,B 0,C 180,E1 -19921.157,E2 -19921.157} C_VEL
LIN {X 0,Y 253.91,Z 482.2,A -85,B 0,C 180,E1 -19923.047,E2 -19923.047} C_VEL
LIN {X 0,Y 256.335,Z 472.359,A -85,B 0,C 180,E1 -19925.609,E2 -19925.609} C_VEL
LIN {X 0,Y 257.185,Z 467.404,A -85,B 0,C 180,E1 -19926.955,E2 -19926.955} C_VEL
LIN {X 0,Y 257.196,Z 465.639,A -85,B 0,C 180,E1 -19927.586,E2 -19927.586} C_VEL
LIN {X 0,Y 256,Z 461.611,A -85,B 0,C 180,E1 -19929.764,E2 -19929.764} C_VEL
LIN {X 0,Y 254.105,Z 456.242,A -85,B 0,C 180,E1 -19934.019,E2 -19934.019} C_VEL
LIN {X 0,Y 253.585,Z 454.679,A -85,B 0,C 180,E1 -19936.143,E2 -19936.143} C_VEL
LIN {X 0,Y 253.236,Z 453.93,A -85,B 0,C 180,E1 -19938.532,E2 -19938.532} C_VEL
LIN {X 0,Y 253.087,Z 454.331,A -85,B 0,C 180,E1 -19941.036,E2 -19941.036} C_VEL
LIN {X 0,Y 253.394,Z 456.259,A -85,B 0,C 180,E1 -19944.377,E2 -19944.377} C_VEL
LIN {X 0,Y 253.631,Z 458.249,A -85,B 0,C 180,E1 -19946.345,E2 -19946.345} C_VEL
LIN {X 0,Y 253.736,Z 460.937,A -85,B 0,C 180,E1 -19948.247,E2 -19948.247} C_VEL
LIN {X 0,Y 253.388,Z 465.678,A -85,B 0,C 180,E1 -19950.909,E2 -19950.909} C_VEL
LIN {X 0,Y 252.658,Z 470.922,A -85,B 0,C 180,E1 -19953.573,E2 -19953.573} C_VEL
LIN {X 0,Y 251.243,Z 476.104,A -85,B 0,C 180,E1 -19956.071,E2 -19956.071} C_VEL
LIN {X 0,Y 250.593,Z 477.806,A -85,B 0,C 180,E1 -19956.881,E2 -19956.881} C_VEL
LIN {X 0,Y 246.068,Z 483.358,A -85,B 0,C 180,E1 -19959.083,E2 -19959.083} C_VEL
LIN {X 0,Y 241.909,Z 487.592,A -85,B 0,C 180,E1 -19961.363,E2 -19961.363} C_VEL
LIN {X 0,Y 239.422,Z 489.667,A -85,B 0,C 180,E1 -19962.93,E2 -19962.93} C_VEL
LIN {X 0,Y 237.123,Z 491.218,A -85,B 0,C 180,E1 -19964.529,E2 -19964.529} C_VEL
LIN {X 0,Y 235.04,Z 492.234,A -85,B 0,C 180,E1 -19966.16,E2 -19966.16} C_VEL
LIN {X 0,Y 233.113,Z 492.717,A -85,B 0,C 180,E1 -19967.817,E2 -19967.817} C_VEL
LIN {X 0,Y 231.314,Z 492.69,A -85,B 0,C 180,E1 -19969.496,E2 -19969.496} C_VEL
LIN {X 0,Y 229.881,Z 492.081,A -85,B 0,C 180,E1 -19971.207,E2 -19971.207} C_VEL
LIN {X 0,Y 228.702,Z 490.909,A -85,B 0,C 180,E1 -19972.939,E2 -19972.939} C_VEL
LIN {X 0,Y 227.382,Z 488.115,A -85,B 0,C 180,E1 -19975.568,E2 -19975.568} C_VEL
LIN {X 0,Y 226.603,Z 483.963,A -85,B 0,C 180,E1 -19978.223,E2 -19978.223} C_VEL
LIN {X 0,Y 226.311,Z 478.297,A -85,B 0,C 180,E1 -19980.89,E2 -19980.89} C_VEL
LIN {X 0,Y 226.457,Z 470.939,A -85,B 0,C 180,E1 -19983.559,E2 -19983.559} C_VEL
LIN {X 0,Y 226.937,Z 463.182,A -85,B 0,C 180,E1 -19985.777,E2 -19985.777} C_VEL
LIN {X 0,Y 227.257,Z 453.59,A -85,B 0,C 180,E1 -19987.952,E2 -19987.952} C_VEL
LIN {X 0,Y 227.742,Z 443.538,A -85,B 0,C 180,E1 -19989.772,E2 -19989.772} C_VEL
LIN {X 0,Y 228.158,Z 434.478,A -85,B 0,C 180,E1 -19991.1,E2 -19991.1} C_VEL
LIN {X 0,Y 226.863,Z 422,A -85,B 0,C 180,E1 -19992.524,E2 -19992.524} C_VEL
LIN {X 0,Y 226.486,Z 416.594,A -85,B 0,C 180,E1 -19993.058,E2 -19993.058} C_VEL
LIN {X 0,Y 226.813,Z 410.008,A -85,B 0,C 180,E1 -19998.051,E2 -19998.051} C_VEL
LIN {X 0,Y 227.285,Z 403.954,A -85,B 0,C 180,E1 -20002.737,E2 -20002.737} C_VEL
LIN {X 0,Y 227.877,Z 397.869,A -85,B 0,C 180,E1 -20007.556,E2 -20007.556} C_VEL
LIN {X 0,Y 228.354,Z 392.912,A -85,B 0,C 180,E1 -20011.548,E2 -20011.548} C_VEL
LIN {X 0,Y 228.178,Z 392.053,A -85,B 0,C 180,E1 -20012.355,E2 -20012.355} C_VEL
LIN {X 0,Y 227.915,Z 392.094,A -85,B 0,C 180,E1 -20016.703,E2 -20016.703} C_VEL
LIN {X 0,Y 227.829,Z 392.105,A -85,B 0,C 180,E1 -20020.377,E2 -20020.377} C_VEL
LIN {X 0,Y 227.838,Z 392.103,A -85,B 0,C 180,E1 -20025.192,E2 -20025.192} C_VEL
LIN {X 0,Y 227.829,Z 392.102,A -85,B 0,C 180,E1 -20029.624,E2 -20029.624} C_VEL
LIN {X 0,Y 227.882,Z 392.097,A -85,B 0,C 180,E1 -20034.128,E2 -20034.128} C_VEL
LIN {X 0,Y 227.873,Z 392.101,A -85,B 0,C 180,E1 -20038.378,E2 -20038.378} C_VEL
LIN {X 0,Y 227.888,Z 392.099,A -85,B 0,C 180,E1 -20042.445,E2 -20042.445} C_VEL
LIN {X 0,Y 227.918,Z 392.095,A -85,B 0,C 180,E1 -20046.368,E2 -20046.368} C_VEL
LIN {X 0,Y 227.946,Z 392.09,A -85,B 0,C 180,E1 -20050.175,E2 -20050.175} C_VEL
LIN {X 0,Y 228.061,Z 392.076,A -85,B 0,C 180,E1 -20053.898,E2 -20053.898} C_VEL
LIN {X 0,Y 228.076,Z 392.07,A -85,B 0,C 180,E1 -20057.543,E2 -20057.543} C_VEL
LIN {X 0,Y 228.271,Z 392.049,A -85,B 0,C 180,E1 -20061.144,E2 -20061.144} C_VEL
LIN {X 0,Y 228.327,Z 392.041,A -85,B 0,C 180,E1 -20062.928,E2 -20062.928} C_VEL
LIN {X 0,Y 228.557,Z 392.015,A -85,B 0,C 180,E1 -20068.238,E2 -20068.238} C_VEL
LIN {X 0,Y 228.558,Z 392.015,A -85,B 0,C 180,E1 -20071.762,E2 -20071.762} C_VEL
LIN {X 0,Y 228.357,Z 392.038,A -85,B 0,C 180,E1 -20077.071,E2 -20077.071} C_VEL
LIN {X 0,Y 228.166,Z 392.061,A -85,B 0,C 180,E1 -20080.65,E2 -20080.65} C_VEL
LIN {X 0,Y 228.068,Z 392.074,A -85,B 0,C 180,E1 -20084.272,E2 -20084.272} C_VEL
LIN {X 0,Y 228.01,Z 392.083,A -85,B 0,C 180,E1 -20087.953,E2 -20087.953} C_VEL
LIN {X 0,Y 227.963,Z 392.085,A -85,B 0,C 180,E1 -20092.348,E2 -20092.348} C_VEL
LIN {X 0,Y 227.945,Z 392.089,A -85,B 0,C 180,E1 -20096.602,E2 -20096.602} C_VEL
LIN {X 0,Y 227.91,Z 392.091,A -85,B 0,C 180,E1 -20100.296,E2 -20100.296} C_VEL
LIN {X 0,Y 227.892,Z 392.098,A -85,B 0,C 180,E1 -20103.718,E2 -20103.718} C_VEL
LIN {X 0,Y 227.872,Z 392.095,A -85,B 0,C 180,E1 -20108.086,E2 -20108.086} C_VEL
LIN {X 0,Y 227.81,Z 392.107,A -85,B 0,C 180,E1 -20112.743,E2 -20112.743} C_VEL
LIN {X 0,Y 227.807,Z 392.107,A -85,B 0,C 180,E1 -20117.256,E2 -20117.256} C_VEL
LIN {X 0,Y 227.845,Z 392.102,A -85,B 0,C 180,E1 -20121.909,E2 -20121.909} C_VEL
LIN {X 0,Y 227.88,Z 392.095,A -85,B 0,C 180,E1 -20126.377,E2 -20126.377} C_VEL
LIN {X 0,Y 227.921,Z 392.093,A -85,B 0,C 180,E1 -20130.438,E2 -20130.438} C_VEL
LIN {X 0,Y 227.931,Z 392.089,A -85,B 0,C 180,E1 -20134.426,E2 -20134.426} C_VEL
LIN {X 0,Y 227.964,Z 392.087,A -85,B 0,C 180,E1 -20138.287,E2 -20138.287} C_VEL
LIN {X 0,Y 228.037,Z 392.078,A -85,B 0,C 180,E1 -20142.825,E2 -20142.825} C_VEL
LIN {X 0,Y 228.097,Z 392.07,A -85,B 0,C 180,E1 -20147.544,E2 -20147.544} C_VEL
LIN {X 0,Y 228.327,Z 392.039,A -85,B 0,C 180,E1 -20151.147,E2 -20151.147} C_VEL
LIN {X 0,Y 228.36,Z 392.039,A -85,B 0,C 180,E1 -20152.929,E2 -20152.929} C_VEL
LIN {X 0,Y 228.557,Z 392.014,A -85,B 0,C 180,E1 -20158.238,E2 -20158.238} C_VEL
LIN {X 0,Y 228.559,Z 392.012,A -85,B 0,C 180,E1 -20161.762,E2 -20161.762} C_VEL
LIN {X 0,Y 228.36,Z 392.036,A -85,B 0,C 180,E1 -20167.071,E2 -20167.071} C_VEL
LIN {X 0,Y 228.173,Z 392.062,A -85,B 0,C 180,E1 -20170.65,E2 -20170.65} C_VEL
LIN {X 0,Y 228.059,Z 392.077,A -85,B 0,C 180,E1 -20176.102,E2 -20176.102} C_VEL
LIN {X 0,Y 227.944,Z 392.09,A -85,B 0,C 180,E1 -20179.825,E2 -20179.825} C_VEL
LIN {X 0,Y 227.915,Z 392.094,A -85,B 0,C 180,E1 -20183.632,E2 -20183.632} C_VEL
LIN {X 0,Y 227.881,Z 392.097,A -85,B 0,C 180,E1 -20187.556,E2 -20187.556} C_VEL
LIN {X 0,Y 227.87,Z 392.1,A -85,B 0,C 180,E1 -20191.622,E2 -20191.622} C_VEL
LIN {X 0,Y 227.901,Z 392.096,A -85,B 0,C 180,E1 -20195.868,E2 -20195.868} C_VEL
LIN {X 0,Y 227.835,Z 392.103,A -85,B 0,C 180,E1 -20200.375,E2 -20200.375} C_VEL
LIN {X 0,Y 227.926,Z 392.093,A -85,B 0,C 180,E1 -20205.744,E2 -20205.744} C_VEL
LIN {X 0,Y 227.981,Z 392.269,A -85,B 0,C 180,E1 -20206.165,E2 -20206.165} C_VEL
LIN {X 0,Y 229.618,Z 400.842,A -85,B 0,C 180,E1 -20211.2,E2 -20211.2} C_VEL
LIN {X 0,Y 231.488,Z 409.544,A -85,B 0,C 180,E1 -20216.064,E2 -20216.064} C_VEL
LIN {X 0,Y 232.394,Z 414.015,A -85,B 0,C 180,E1 -20218.489,E2 -20218.489} C_VEL
LIN {X 0,Y 231.249,Z 418.675,A -85,B 0,C 180,E1 -20220.905,E2 -20220.905} C_VEL
LIN {X 0,Y 228.769,Z 429.34,A -85,B 0,C 180,E1 -20226.461,E2 -20226.461} C_VEL
LIN {X 0,Y 227.957,Z 434.566,A -85,B 0,C 180,E1 -20229.214,E2 -20229.214} C_VEL
LIN {X 0,Y 227.331,Z 436.143,A -85,B 0,C 180,E1 -20229.779,E2 -20229.779} C_VEL
LIN {X 0,Y 225.586,Z 438.879,A -85,B 0,C 180,E1 -20230.304,E2 -20230.304} C_VEL
LIN {X 0,Y 221.949,Z 444.691,A -85,B 0,C 180,E1 -20230.837,E2 -20230.837} C_VEL
LIN {X 0,Y 220.778,Z 448.487,A -85,B 0,C 180,E1 -20231.166,E2 -20231.166} C_VEL
LIN {X 0,Y 220.641,Z 454.411,A -85,B 0,C 180,E1 -20231.741,E2 -20231.741} C_VEL
LIN {X 0,Y 221.565,Z 462.255,A -85,B 0,C 180,E1 -20232.619,E2 -20232.619} C_VEL
LIN {X 0,Y 222.281,Z 471.977,A -85,B 0,C 180,E1 -20233.939,E2 -20233.939} C_VEL
LIN {X 0,Y 221.647,Z 482.453,A -85,B 0,C 180,E1 -20235.775,E2 -20235.775} C_VEL
LIN {X 0,Y 221.138,Z 490.984,A -85,B 0,C 180,E1 -20237.613,E2 -20237.613} C_VEL
LIN {X 0,Y 220.709,Z 499.662,A -85,B 0,C 180,E1 -20239.914,E2 -20239.914} C_VEL
LIN {X 0,Y 220.598,Z 507.98,A -85,B 0,C 180,E1 -20242.679,E2 -20242.679} C_VEL
LIN {X 0,Y 220.672,Z 512.458,A -85,B 0,C 180,E1 -20244.517,E2 -20244.517} C_VEL
LIN {X 0,Y 220.744,Z 517.855,A -85,B 0,C 180,E1 -20247.263,E2 -20247.263} C_VEL
LIN {X 0,Y 220.601,Z 521.773,A -85,B 0,C 180,E1 -20250,E2 -20250} C_VEL
LIN {X 0,Y 220.285,Z 523.644,A -85,B 0,C 180,E1 -20251.828,E2 -20251.828} C_VEL
LIN {X 0,Y 219.787,Z 525.024,A -85,B 0,C 180,E1 -20253.667,E2 -20253.667} C_VEL
LIN {X 0,Y 219.334,Z 526.38,A -85,B 0,C 180,E1 -20256.628,E2 -20256.628} C_VEL
LIN {X 0,Y 219.287,Z 526.739,A -85,B 0,C 180,E1 -20259.221,E2 -20259.221} C_VEL
LIN {X 0,Y 219.953,Z 526.057,A -85,B 0,C 180,E1 -20262.925,E2 -20262.925} C_VEL
LIN {X 0,Y 221.912,Z 523.935,A -85,B 0,C 180,E1 -20266.561,E2 -20266.561} C_VEL
LIN {X 0,Y 224.874,Z 520.398,A -85,B 0,C 180,E1 -20270.108,E2 -20270.108} C_VEL
LIN {X 0,Y 229.034,Z 515.306,A -85,B 0,C 180,E1 -20273.51,E2 -20273.51} C_VEL
LIN {X 0,Y 232.936,Z 510.396,A -85,B 0,C 180,E1 -20275.944,E2 -20275.944} C_VEL
LIN {X 0,Y 237.366,Z 504.386,A -85,B 0,C 180,E1 -20278.277,E2 -20278.277} C_VEL
LIN {X 0,Y 243.247,Z 495.864,A -85,B 0,C 180,E1 -20280.853,E2 -20280.853} C_VEL
LIN {X 0,Y 246.821,Z 488.896,A -85,B 0,C 180,E1 -20282.752,E2 -20282.752} C_VEL
LIN {X 0,Y 249.934,Z 480.432,A -85,B 0,C 180,E1 -20285.123,E2 -20285.123} C_VEL
LIN {X 0,Y 251.983,Z 473.013,A -85,B 0,C 180,E1 -20287.235,E2 -20287.235} C_VEL
LIN {X 0,Y 252.373,Z 471.221,A -85,B 0,C 180,E1 -20287.782,E2 -20287.782} C_VEL
LIN {X 0,Y 251.644,Z 467.172,A -85,B 0,C 180,E1 -20289.968,E2 -20289.968} C_VEL
LIN {X 0,Y 250.343,Z 463.202,A -85,B 0,C 180,E1 -20293.121,E2 -20293.121} C_VEL
LIN {X 0,Y 249.811,Z 461.261,A -85,B 0,C 180,E1 -20295.305,E2 -20295.305} C_VEL
LIN {X 0,Y 249.441,Z 460.146,A -85,B 0,C 180,E1 -20297.453,E2 -20297.453} C_VEL
LIN {X 0,Y 249.174,Z 459.874,A -85,B 0,C 180,E1 -20299.601,E2 -20299.601} C_VEL
LIN {X 0,Y 249.009,Z 460.676,A -85,B 0,C 180,E1 -20302.211,E2 -20302.211} C_VEL
LIN {X 0,Y 249.054,Z 462.496,A -85,B 0,C 180,E1 -20304.92,E2 -20304.92} C_VEL
LIN {X 0,Y 249.056,Z 463.838,A -85,B 0,C 180,E1 -20306.309,E2 -20306.309} C_VEL
